(* IEC 61131-3 sources: elnaProjects/ElpcLogic/PomarKc7Changed/build_USO_ecl (part 6) *)

  StrAlg.status :=  SHL(BYTE_TO_DWORD(source_for_Status), 29)
  			OR SHL(BYTE_TO_DWORD(cmd_for_Status), 26)
  			OR SHL(BYTE_TO_DWORD(command_error_for_Status), 23)
  			OR SHL(BOOL_TO_DWORD(StrAlg.OpcCommandsDisabled ), 21)
  			OR SHL(BOOL_TO_DWORD(StrAlg.hasError),4)
  			OR SHL(BOOL_TO_DWORD(StrAlg.CanRun),2)
  			OR SHL(BOOL_TO_DWORD(StrAlg.isEnded),1)
  			OR BOOL_TO_DWORD(StrAlg.isRuning);
END_FUNCTION_BLOCK

FUNCTION_BLOCK fb_AutoTenAlg
  VAR_IN_OUT
    StrAlg : struct_Alg;
    PNS : struct_Switch;
    TEN : struct_Switch;
  END_VAR
  VAR_INPUT
    T_masla : struct_AI;
    Uroven_masla : struct_AI;
    offTemperature : struct_AnalogParametr;
  END_VAR
  VAR
    _sunpackerCommand : fb_sunpackerCommand;
    _statusAi : TYPE_StatusAi;
    _statusDualInput : TYPE_statusDualInput;
    _commandDualInput : TYPE_commandDualInput;
    source : BYTE;
    cmd : BYTE;
    lastCmd : BYTE;
    source_for_Status : BYTE;
    cmd_for_Status : BYTE;
    command_error_for_Status : BYTE;
    resetCmdTimer : TON;
    resetCmdTimerPriznak : BOOL;
    onInit : BOOL;
  END_VAR

  IF NOT onInit THEN
  StrAlg.inCanRun:=TRUE;
  onInit:=TRUE;
  END_IF;

  IF StrAlg.isRuning THEN

  IF ((T_masla.interval >= _statusAi.normal) AND (T_masla.value > offTemperature.Value)) OR
  ((Uroven_masla.interval >= _statusAi.normal) AND (Uroven_masla.value < Uroven_masla.LA)) OR
  (PNS.onStatus=_statusDualInput.STATUS_OFF) THEN

        TEN.inOpcCommandsDisabled:=TRUE;

  	IF TEN.onStatus = _statusDualInput.STATUS_ON THEN
            TEN.inCommand_Alg:=BYTE_TO_WORD(_commandDualInput.CMD_OFF);
  	END_IF;

  ELSIF PNS.onStatus = _statusDualInput.STATUS_ON THEN
        TEN.inOpcCommandsDisabled:=FALSE;
  END_IF;

  END_IF;

  StrAlg.CanRun := StrAlg.inCanRun;
  StrAlg.hasError := TEN.CommandFault OR (T_masla.interval < _statusAi.normal) OR (Uroven_masla.interval < _statusAi.normal);

  StrAlg.OpcCommandsDisabled := StrAlg.inOpcCommandsDisabled;

  (* ---- Если управление с ВУ заблокировано, то  передаем команду из алгоритма ---- *)
  IF StrAlg.inOpcCommandsDisabled THEN
  	StrAlg.inCommand := StrAlg.inCommand_Alg;
  ELSE (* иначе передаем команду с АРМа*)
  	StrAlg.inCommand := StrAlg.inCommand_ARM;
  END_IF;

  _sunpackerCommand(command := StrAlg.inCommand);
  	source := _sunpackerCommand.source;
  	cmd := _sunpackerCommand.cmd;

  IF cmd <> 0 AND lastCmd <> cmd AND (((NOT StrAlg.opcCommandsDisabled) AND source > 0) OR source = 0) then
  	CASE BYTE_TO_INT(cmd) OF
  		(*cmdRun*) 1: 	IF StrAlg.CanRun AND NOT StrAlg.hasError THEN
  					StrAlg.isRuning := TRUE;
  					StrAlg.isEnded := FALSE;
  					(*StrAlg.hasError := FALSE;*)

                                                    (*****************       OnRun       *****************)
                                                    IF StrAlg.inOpcCommandsDisabled THEN
  		                              StrAlg.inOpcCommandsDisabled:=FALSE;
                                                    END_IF;
  					cmd_for_Status := cmd;
  					source_for_Status := source;
  					command_error_for_Status := 0;
  				ELSE
  					StrAlg.isRuning := FALSE;
  					StrAlg.isEnded := FALSE;
  					(*StrAlg.hasError 	:= FALSE;*)

  					cmd_for_Status := 0;
  					source_for_Status := source;
  					command_error_for_Status := cmd;
  				END_IF;
  		(*cmdReset*) 2: 	StrAlg.isRuning := FALSE;
  				StrAlg.isEnded := FALSE;
  				(*StrAlg.hasError 	:= FALSE;*)

                                          (*****************       OnReset       *****************)
                                          TEN.inOpcCommandsDisabled:=TRUE;
                                          TEN.inCommand_Alg:=BYTE_TO_WORD(_commandDualInput.CMD_OFF);

  				cmd_for_Status := cmd;
  				source_for_Status := source;
  				command_error_for_Status := 0;
  	END_CASE;
  	resetCmdTimer(IN := false);
  	resetCmdTimerPriznak := TRUE;
  END_IF;
  lastCmd := cmd;

  resetCmdTimer(IN := resetCmdTimerPriznak, PT := T#5S);
  IF resetCmdTimer.Q THEN
  	resetCmdTimerPriznak := FALSE;
  	source_for_Status := 0;
  	cmd_for_Status := 0;
  	command_error_for_Status := 0;
  END_IF;

  (*TODO: TYPE PROGRAM CODE HERE*)
  StrAlg.status :=  SHL(BYTE_TO_DWORD(source_for_Status), 29)
  			OR SHL(BYTE_TO_DWORD(cmd_for_Status), 26)
  			OR SHL(BYTE_TO_DWORD(command_error_for_Status), 23)
  			OR SHL(BOOL_TO_DWORD(StrAlg.OpcCommandsDisabled ), 21)
  			OR SHL(BOOL_TO_DWORD(StrAlg.hasError),4)
  			OR SHL(BOOL_TO_DWORD(StrAlg.CanRun),2)
  			OR SHL(BOOL_TO_DWORD(StrAlg.isEnded),1)
  			OR BOOL_TO_DWORD(StrAlg.isRuning);
END_FUNCTION_BLOCK

FUNCTION_BLOCK fb_AutoPnsAlg
  VAR_IN_OUT
    StrAlg : struct_Alg;
    Nasos : struct_Switch;
  END_VAR
  VAR_INPUT
    diPlow : struct_singleSignal;
    Poil : struct_AI;
    Ust_Run : struct_AnalogParametr;
    Ust_Stop : struct_AnalogParametr;
  END_VAR
  VAR
    _sunpackerCommand : fb_sunpackerCommand;
    _statusAi : TYPE_StatusAi;
    _statusDualInput : TYPE_statusDualInput;
    _commandDualInput : TYPE_commandDualInput;
    source : BYTE;
    cmd : BYTE;
    lastCmd : BYTE;
    source_for_Status : BYTE;
    cmd_for_Status : BYTE;
    command_error_for_Status : BYTE;
    resetCmdTimer : TON;
    resetCmdTimerPriznak : BOOL;
    onInit : BOOL;
    onTrig : R_TRIG;
    offTrig : R_TRIG;
    waitOn : TON;
    waitOff : TON;
  END_VAR
  VAR_EXTERNAL
    AlgTimers : struct_AlgTimers;
  END_VAR

  IF NOT onInit THEN
  StrAlg.inOpcCommandsDisabled:=TRUE;
  StrAlg.inCanRun:=TRUE;
  onInit:=TRUE;
  END_IF;

  IF StrAlg.isRuning THEN

  StrAlg.hasError := Nasos.CommandFault OR (Poil.interval < _statusAi.normal OR NOT diPlow.reliability);

      IF (Poil.Interval >= _statusAi.normal) THEN
      waitOn(IN:=Poil.Value <= Ust_Run.value OR diPlow.q, PT := T#1S);
      waitOff(IN:= Poil.Value >= Ust_Stop.value, PT := T#300S);

      ELSE
      waitOn(IN:=diPlow.Q, PT := T#1S);
      END_IF;

  onTrig(CLK:=waitOn.Q);
  offTrig(CLK:=waitOff.Q);
      IF (Poil.Value>=Ust_Stop.value) AND Nasos.inopcCommandsDisabled THEN
          Nasos.inopcCommandsDisabled:=FALSE;
      END_IF;

      IF onTrig.Q THEN
      Nasos.inopcCommandsDisabled:=TRUE;
      Nasos.inCommand_Alg:=BYTE_TO_WORD(_commandDualInput.CMD_ON);
      END_IF;

      IF offTrig.Q THEN
          IF NOT (Nasos.onStatus=_statusDualInput.STATUS_OFF) THEN
          Nasos.inopcCommandsDisabled:=TRUE;
          Nasos.inCommand_Alg:=BYTE_TO_WORD(_commandDualInput.CMD_OFF);
          END_IF;
      END_IF;

  AlgTimers.AutoPns_OnTimer:=UDINT_TO_UINT(TIME_TO_UDINT(waitOn.PT - waitOn.ET)/1000);
  AlgTimers.AutoPns_OffTimer:=UDINT_TO_UINT(TIME_TO_UDINT(waitOff.PT -waitOff.ET)/1000);

  END_IF;

  StrAlg.CanRun := StrAlg.inCanRun;

  StrAlg.OpcCommandsDisabled := StrAlg.inOpcCommandsDisabled;

  (* ---- Если управление с ВУ заблокировано, то  передаем команду из алгоритма ---- *)
  IF StrAlg.inOpcCommandsDisabled THEN
  	StrAlg.inCommand := StrAlg.inCommand_Alg;
  ELSE (* иначе передаем команду с АРМа*)
  	StrAlg.inCommand := StrAlg.inCommand_ARM;
  END_IF;

  _sunpackerCommand(command := StrAlg.inCommand);
  	source := _sunpackerCommand.source;
  	cmd := _sunpackerCommand.cmd;

  IF cmd <> 0 AND lastCmd <> cmd AND (((NOT StrAlg.opcCommandsDisabled) AND source > 0) OR source = 0) then
  	CASE BYTE_TO_INT(cmd) OF
  		(*cmdRun*) 1: 	IF (StrAlg.CanRun) THEN
  					StrAlg.isRuning := TRUE;
  					StrAlg.isEnded := FALSE;
  					StrAlg.hasError := FALSE;
  					(*****************       OnRun       *****************)

  					cmd_for_Status := cmd;
  					source_for_Status := source;
  					command_error_for_Status := 0;
  				ELSE
  					StrAlg.isRuning := FALSE;
  					StrAlg.isEnded := FALSE;
  					StrAlg.hasError 	:= FALSE;

  					cmd_for_Status := 0;
  					source_for_Status := source;
  					command_error_for_Status := cmd;
  				END_IF;
  		(*cmdReset*) 2: 	StrAlg.isRuning := FALSE;
  				StrAlg.isEnded := FALSE;
  				StrAlg.hasError 	:= FALSE;

                                           (*****************       OnReset       *****************)
                                          waitOn(in:=FALSE);
                                          waitOff(in:=FALSE);
                                          AlgTimers.AutoPns_OffTimer:=UDINT_TO_UINT(TIME_TO_UDINT(waitOff.pt -waitOff.ET)/1000);

  				cmd_for_Status := cmd;
  				source_for_Status := source;
  				command_error_for_Status := 0;
  	END_CASE;
  	resetCmdTimer(IN := false);
  	resetCmdTimerPriznak := TRUE;
  END_IF;
  lastCmd := cmd;

  resetCmdTimer(IN := resetCmdTimerPriznak, PT := T#5S);
  IF resetCmdTimer.Q THEN
  	resetCmdTimerPriznak := FALSE;
  	source_for_Status := 0;
  	cmd_for_Status := 0;
  	command_error_for_Status := 0;
  END_IF;

  (*TODO: TYPE PROGRAM CODE HERE*)
  StrAlg.status :=  SHL(BYTE_TO_DWORD(source_for_Status), 29)
  			OR SHL(BYTE_TO_DWORD(cmd_for_Status), 26)
  			OR SHL(BYTE_TO_DWORD(command_error_for_Status), 23)
  			OR SHL(BOOL_TO_DWORD(StrAlg.OpcCommandsDisabled ), 21)
  			OR SHL(BOOL_TO_DWORD(StrAlg.hasError),4)
  			OR SHL(BOOL_TO_DWORD(StrAlg.CanRun),2)
  			OR SHL(BOOL_TO_DWORD(StrAlg.isEnded),1)
  			OR BOOL_TO_DWORD(StrAlg.isRuning);
END_FUNCTION_BLOCK

FUNCTION_BLOCK fb_AutoAvomAlg
  VAR_IN_OUT
    StrAlg : struct_Alg;
    im1 : struct_Switch;
    im2 : struct_Switch;
  END_VAR
  VAR_INPUT
    ai : struct_AI;
  END_VAR
  VAR_IN_OUT
    on1Temperature : struct_AnalogParametr;
    on2Temperature : struct_AnalogParametr;
    hystereses : struct_AnalogParametr;
  END_VAR
  VAR
    _sunpackerCommand : fb_sunpackerCommand;
    _statusAi : TYPE_StatusAi;
    _statusDualInput : TYPE_statusDualInput;
    _commandDualInput : TYPE_commandDualInput;
    source : BYTE;
    cmd : BYTE;
    lastCmd : BYTE;
    source_for_Status : BYTE;
    cmd_for_Status : BYTE;
    command_error_for_Status : BYTE;
    resetCmdTimer : TON;
    resetCmdTimerPriznak : BOOL;
    onInit : BOOL;
  END_VAR

  (*
  IF NOT onInit THEN
  StrAlg.inCanRun:=TRUE;
  onInit:=TRUE;
  END_IF;
  *)

  IF StrAlg.isRuning THEN

  StrAlg.hasError := im1.CommandFault OR im2.CommandFault OR (ai.interval<_statusAi.normal);

      IF (ai.interval>=_statusAi.normal) THEN

            IF (ai.value>= on1Temperature.Value) THEN
                IF im1.onStatus <> _statusDualInput.STATUS_ON THEN
  	       im1.inCommand_Alg:=BYTE_TO_WORD(_commandDualInput.CMD_ON); (*cmd_on*)
                END_IF;
            END_IF;

            IF  ai.value < (on1Temperature.Value - hystereses.Value) THEN
                IF im1.onStatus <> _statusDualInput.STATUS_OFF THEN
  	       im1.inCommand_Alg:=BYTE_TO_WORD(_commandDualInput.CMD_OFF);
                END_IF;
            END_IF;

             IF (ai.value>= on2Temperature.Value) THEN
                IF im2.onStatus <> _statusDualInput.STATUS_ON THEN
  	       im2.inCommand_Alg:=BYTE_TO_WORD(_commandDualInput.CMD_ON); (*cmd_on*)
                END_IF;
            END_IF;

            IF  ai.value < (on2Temperature.Value - hystereses.Value) THEN
                IF im2.onStatus <> _statusDualInput.STATUS_OFF THEN
  	       im2.inCommand_Alg:=BYTE_TO_WORD(_commandDualInput.CMD_OFF);
                END_IF;
            END_IF;
       END_IF;

  END_IF;

  StrAlg.CanRun := StrAlg.inCanRun;

  StrAlg.OpcCommandsDisabled := StrAlg.inOpcCommandsDisabled;

  (* ---- Если управление с ВУ заблокировано, то  передаем команду из алгоритма ---- *)
  IF StrAlg.inOpcCommandsDisabled THEN
  	StrAlg.inCommand := StrAlg.inCommand_Alg;
  ELSE (* иначе передаем команду с АРМа*)
  	StrAlg.inCommand := StrAlg.inCommand_ARM;
  END_IF;

  _sunpackerCommand(command := StrAlg.inCommand);
  	source := _sunpackerCommand.source;
  	cmd := _sunpackerCommand.cmd;

  IF cmd <> 0 AND lastCmd <> cmd AND (((NOT StrAlg.opcCommandsDisabled) AND source > 0) OR source = 0) then
  	CASE BYTE_TO_INT(cmd) OF
  		(*cmdRun*) 1: 	IF (StrAlg.CanRun) THEN
  					StrAlg.isRuning := TRUE;
  					StrAlg.isEnded := FALSE;
  					StrAlg.hasError := FALSE;
                                                    StrAlg.inOpcCommandsDisabled:=FALSE;
  					im1.inOpcCommandsDisabled:=TRUE;
                                                    im2.inOpcCommandsDisabled:=TRUE;
  					cmd_for_Status := cmd;
  					source_for_Status := source;
  					command_error_for_Status := 0;
  				ELSE
  					StrAlg.isRuning := FALSE;
  					StrAlg.isEnded := FALSE;
  					StrAlg.hasError 	:= FALSE;

  					cmd_for_Status := 0;
  					source_for_Status := source;
  					command_error_for_Status := cmd;
  				END_IF;
  		(*cmdReset*) 2: 	StrAlg.isRuning := FALSE;
  				StrAlg.isEnded := FALSE;
  				StrAlg.hasError 	:= FALSE;
                                          StrAlg.inOpcCommandsDisabled:=FALSE;
                                          im1.inOpcCommandsDisabled:=FALSE;
                                          im2.inOpcCommandsDisabled:=FALSE;
                                          im1.inCommand_Alg:=0;
                                          im2.inCommand_Alg:=0;
  				cmd_for_Status := cmd;
  				source_for_Status := source;
  				command_error_for_Status := 0;
  	END_CASE;
  	resetCmdTimer(IN := false);
  	resetCmdTimerPriznak := TRUE;
  END_IF;
  lastCmd := cmd;

  resetCmdTimer(IN := resetCmdTimerPriznak, PT := T#5S);
  IF resetCmdTimer.Q THEN
  	resetCmdTimerPriznak := FALSE;
  	source_for_Status := 0;
  	cmd_for_Status := 0;
  	command_error_for_Status := 0;
  END_IF;

  (*TODO: TYPE PROGRAM CODE HERE*)
  StrAlg.status :=  SHL(BYTE_TO_DWORD(source_for_Status), 29)
  			OR SHL(BYTE_TO_DWORD(cmd_for_Status), 26)
  			OR SHL(BYTE_TO_DWORD(command_error_for_Status), 23)
  			OR SHL(BOOL_TO_DWORD(StrAlg.OpcCommandsDisabled ), 21)
  			OR SHL(BOOL_TO_DWORD(StrAlg.hasError),4)
  			OR SHL(BOOL_TO_DWORD(StrAlg.CanRun),2)
  			OR SHL(BOOL_TO_DWORD(StrAlg.isEnded),1)
  			OR BOOL_TO_DWORD(StrAlg.isRuning);
END_FUNCTION_BLOCK

FUNCTION_BLOCK fb_vibegPNSAlg
  VAR_IN_OUT
    StrAlg : struct_Alg;
  END_VAR
  VAR
    autoPnsOff : struct_PhaseAlgoritm;
    waitVibeg : struct_PhaseAlgoritm;
    pnsOff : struct_PhaseAlgoritm;
    vibegEnd : struct_PhaseAlgoritm;
  END_VAR
  VAR_IN_OUT
    algContinue : struct_Question;
  END_VAR
  VAR
    fb_autoPnsOff : fb_ph_algoritm;
    fb_waitVibeg : fb_ph_Timer;
    fb_algContinue : fb_Question;
    fb_pnsOff : fb_ph_Switch;
    fb_vibegEnd : fb_ph_CustomPhase;
    _sunpackerCommand : fb_sunpackerCommand;
    _statusAi : TYPE_StatusAi;
    _Answers : TYPE_Answers;
    _statusDualInput : TYPE_statusDualInput;
    _DualStateImAction : TYPE_DualStateImAction;
    _PhaseAlgoritmAction : TYPE_PhaseAlgoritmAction;
    source : BYTE;
    cmd : BYTE;
    lastCmd : BYTE;
    source_for_Status : BYTE;
    cmd_for_Status : BYTE;
    command_error_for_Status : BYTE;
    resetCmdTimer : TON;
    resetCmdTimerPriznak : BOOL;
    onInit : BOOL;
    waitReset : TON;
  END_VAR
  VAR_EXTERNAL
    IM : ImConfig;
    algoritms : AlgoritmsConfig;
    ai : AiConfig;
    protections : ProtectionsConfig;
    AlgTimers : struct_AlgTimers;
  END_VAR

  IF NOT onInit THEN
   fb_autoPnsOff(phaseNumber:=0, act:=_reset, waitCompletion:=FALSE);
    fb_waitVibeg(phaseNumber:=1, delay:=T#300S);
       algContinue.AnswerVariants:=_Answers.ANS_YES;
       fb_pnsOff(phaseNumber:=2, act:=_off);
     fb_vibegEnd(phaseNumber:=14);
  onInit:=TRUE;
  END_IF;

   fb_autoPnsOff(StrPh:=autoPnsOff, alg:=algoritms.autoPns);
    fb_waitVibeg(StrPh:=waitVibeg, timer:=AlgTimers.vibegPNS_Timer);
  fb_algContinue(StrQ:=algContinue);
       fb_pnsOff(StrPh:=pnsOff, Im:=IM.pns);
     fb_vibegEnd(StrPh:=vibegEnd);

  IF StrAlg.isRuning THEN

  StrAlg.hasError := autoPnsOff.error OR pnsOff.error;

      IF IM.pns.onStatus = _statusDualInput.STATUS_ON AND NOT vibegEnd.top THEN

  	runPhase(vibegEnd);
            runPhase(waitVibeg);
            askQuestion(algContinue);

      END_IF;

      IF waitVibeg.top OR (algContinue.answer = _Answers.ANS_YES) THEN
  	vibegEnd.top:=TRUE;
  	resetPhase(waitVibeg);
            resetQuestion(algContinue);

            resetAiProtection(protections.Os_sdvig_nagnetatelja_minus);
            (*resetDiProtection(protections.Vibro_skorost_OP_shesterni_RED_T6);*)

  	(*IM.SingleSignals.P_oil_low.Disabled_Sig:=TRUE;*)
  	ai.Pmasla_posle_GNS.Disabled_LA:=TRUE;
            ai.Pmasla_posle_GNS.Disabled_LW:=TRUE;
            ai.Pmasla_posle_NU.Disabled_LW:=TRUE;
  	runPhase(pnsOff);
      END_IF;

      StrAlg.isEnded:=pnsOff.top;

  END_IF;

  StrAlg.CanRun := StrAlg.inCanRun;
  StrAlg.OpcCommandsDisabled := StrAlg.inOpcCommandsDisabled;

  (* ---- Если управление с ВУ заблокировано, то  передаем команду из алгоритма ---- *)
  IF StrAlg.inOpcCommandsDisabled THEN
  	StrAlg.inCommand := StrAlg.inCommand_Alg;
  ELSE (* иначе передаем команду с АРМа*)
  	StrAlg.inCommand := StrAlg.inCommand_ARM;
  END_IF;

  _sunpackerCommand(command := StrAlg.inCommand);
  	source := _sunpackerCommand.source;
  	cmd := _sunpackerCommand.cmd;

  IF cmd <> 0 AND lastCmd <> cmd AND (((NOT StrAlg.opcCommandsDisabled) AND source > 0) OR source = 0) then
  	CASE BYTE_TO_INT(cmd) OF
  		(*cmdRun*) 1: 	IF (StrAlg.CanRun) THEN
  					StrAlg.isRuning := TRUE;
  					StrAlg.isEnded := FALSE;
  					StrAlg.hasError := FALSE;
  					(*****************       OnRun       *****************)
                                                    runPhase(autoPnsOff);

  					cmd_for_Status := cmd;
  					source_for_Status := source;
  					command_error_for_Status := 0;
  				ELSE
  					StrAlg.isRuning := FALSE;
  					StrAlg.isEnded := FALSE;
  					StrAlg.hasError 	:= FALSE;

  					cmd_for_Status := 0;
  					source_for_Status := source;
  					command_error_for_Status := cmd;
  				END_IF;
  		(*cmdReset*) 2: 	StrAlg.isRuning := FALSE;
  				StrAlg.isEnded := FALSE;
  				StrAlg.hasError 	:= FALSE;

                                           (*****************       OnReset       *****************)
                                         waitReset(IN:=FALSE);
                                         resetPhase(autoPnsOff);
                                         resetPhase(waitVibeg);
                                         resetPhase(vibegEnd);
                                         resetPhase(pnsOff);
                                         resetQuestion(algContinue);

  				cmd_for_Status := cmd;
  				source_for_Status := source;
  				command_error_for_Status := 0;
  	END_CASE;
  	resetCmdTimer(IN := false);
  	resetCmdTimerPriznak := TRUE;
  END_IF;
  lastCmd := cmd;

  resetCmdTimer(IN := resetCmdTimerPriznak, PT := T#5S);
  IF resetCmdTimer.Q THEN
  	resetCmdTimerPriznak := FALSE;
  	source_for_Status := 0;
  	cmd_for_Status := 0;
  	command_error_for_Status := 0;
  END_IF;

  StrAlg.Start:= autoPnsOff.startStatus
              OR waitVibeg.startStatus
              OR pnsOff.startStatus
              OR vibegEnd.startStatus;

  StrAlg.Error:= autoPnsOff.errorStatus
              OR waitVibeg.errorStatus
              OR pnsOff.errorStatus
              OR vibegEnd.errorStatus;

  StrAlg.Top:=   autoPnsOff.topStatus
              OR waitVibeg.topStatus
              OR pnsOff.topStatus
              OR vibegEnd.topStatus;

  (*TODO: TYPE PROGRAM CODE HERE*)
  StrAlg.status :=  SHL(BYTE_TO_DWORD(source_for_Status), 29)
  			OR SHL(BYTE_TO_DWORD(cmd_for_Status), 26)
  			OR SHL(BYTE_TO_DWORD(command_error_for_Status), 23)
  			OR SHL(BOOL_TO_DWORD(StrAlg.OpcCommandsDisabled ), 21)
  			OR SHL(BOOL_TO_DWORD(StrAlg.hasError),4)
  			OR SHL(BOOL_TO_DWORD(StrAlg.CanRun),2)
  			OR SHL(BOOL_TO_DWORD(StrAlg.isEnded),1)
  			OR BOOL_TO_DWORD(StrAlg.isRuning);
END_FUNCTION_BLOCK

FUNCTION_BLOCK fb_AutoNUAlg
  VAR_IN_OUT
    StrAlg : struct_Alg;
    nu1 : struct_OilPump;
    nu2 : struct_OilPump;
  END_VAR
  VAR_INPUT
    dPoil : struct_AI;
  END_VAR
  VAR_IN_OUT
    mainNU : struct_DiscretParametr;
    Lowdp_di : struct_singleSignal;
    Ust_Swap : struct_AnalogParametr;
  END_VAR
  VAR
    _prevMainNU : UINT;
    _sunpackerCommand : fb_sunpackerCommand;
    _statusAi : TYPE_StatusAi;
    _statusDualInput : TYPE_statusDualInput;
    _commandDualInput : TYPE_commandDualInput;
    source : BYTE;
    cmd : BYTE;
    lastCmd : BYTE;
    source_for_Status : BYTE;
    cmd_for_Status : BYTE;
    command_error_for_Status : BYTE;
    resetCmdTimer : TON;
    waitPressure : TON;
    waitPressureTrig : R_TRIG;
    resetCmdTimerPriznak : BOOL;
    onInit : BOOL;
    onStart : BOOL;
  END_VAR
  VAR_EXTERNAL
    NotHasRezervNU : BOOL;
    Reset_HasNU : BOOL;
  END_VAR

  IF NOT onInit THEN
  StrAlg.inCanRun:=TRUE;
  StrAlg.inOpcCommandsDisabled:=TRUE;
  (*nu1.Osnovnoy:=TRUE; nu2.Osnovnoy:=FALSE;*)
  onInit:=TRUE;
  END_IF;

  IF Reset_HasNU THEN
  nu1.inBlocked:=FALSE;
  nu2.inBlocked:=FALSE;
  END_IF;

  NotHasRezervNU:=(nu1.Blocked OR nu2.Blocked);

  IF StrAlg.isRuning THEN

  StrAlg.hasError := nu1.CommandFault OR nu2.CommandFault OR (dPoil.interval<_statusAi.normal);

   IF mainNU.value<>_prevMainNU OR NOT onStart THEN

          CASE mainNU.value OF
  	0: nu1.Osnovnoy:=TRUE; nu2.Osnovnoy:=FALSE;
  	1: nu1.Osnovnoy:=FALSE; nu2.Osnovnoy:=TRUE;

          END_CASE;

      IF  nu1.Osnovnoy AND NOT nu1.Blocked THEN
          nu1.inCommand_Alg:=BYTE_TO_WORD(_commandDualInput.CMD_ON);
      ELSIF NOT NotHasRezervNU THEN
          nu1.inCommand_Alg:=BYTE_TO_WORD(_commandDualInput.CMD_OFF);
      END_IF;

      IF  nu2.Osnovnoy AND NOT nu2.Blocked THEN
          nu2.inCommand_Alg:=BYTE_TO_WORD(_commandDualInput.CMD_ON);
       ELSIF NOT NotHasRezervNU THEN
          nu2.inCommand_Alg:=BYTE_TO_WORD(_commandDualInput.CMD_OFF);
      END_IF;
        onStart:=TRUE;
       _prevMainNU:=mainNU.value;
   END_IF;

    (*IF (nu1.onStatus = _statusDualInput.STATUS_On) OR (nu2.onStatus = _statusDualInput.STATUS_On) THEN*)
      (*Если через 5С насос не нагнал 100кПа масла - он сломался и надо переключить насос*)
      IF dPoil.interval>= _statusAi.NORMAL THEN
            waitPressure(IN:=(dPoil.value<Ust_Swap.Value OR LowdP_DI.q) AND NOT NotHasRezervNU, PT:= T#5S);
      ELSE
  	waitPressure(IN:=(FALSE));
      END_IF;

      waitPressureTrig(CLK:=waitPressure.Q);
      IF waitPressureTrig.Q THEN
  	(*IF nu1.onStatus = _statusDualInput.STATUS_ON THEN*)
             IF mainNU.value = 0 THEN
  		nu1.inBlocked:=TRUE;
                      nu1.inCommand_Alg:=BYTE_TO_WORD(_commandDualInput.CMD_OFF);
  			(*IF 	mainNU.value = 0 THEN*)
                                          setValue(mainNU, 1);
  			(*END_IF;*)
  	END_IF;

  	(*IF nu2.onStatus = _statusDualInput.STATUS_ON THEN*)
            IF mainNU.value = 1 THEN
  		nu2.inBlocked:=TRUE;
                      nu2.inCommand_Alg:=BYTE_TO_WORD(_commandDualInput.CMD_OFF);
  			(*IF 	mainNU.value = 1 THEN*)
  				setValue(mainNU, 0);
  			(*END_IF;*)
  	END_IF;
      END_IF;
   (* END_IF;*)

  END_IF;

  StrAlg.CanRun := StrAlg.inCanRun;

  StrAlg.OpcCommandsDisabled := StrAlg.inOpcCommandsDisabled;

  (* ---- Если управление с ВУ заблокировано, то  передаем команду из алгоритма ---- *)
  IF StrAlg.inOpcCommandsDisabled THEN
  	StrAlg.inCommand := StrAlg.inCommand_Alg;
  ELSE (* иначе передаем команду с АРМа*)
  	StrAlg.inCommand := StrAlg.inCommand_ARM;
  END_IF;

  _sunpackerCommand(command := StrAlg.inCommand);
  	source := _sunpackerCommand.source;
  	cmd := _sunpackerCommand.cmd;

  IF cmd <> 0 AND lastCmd <> cmd AND (((NOT StrAlg.opcCommandsDisabled) AND source > 0) OR source = 0) then
  	CASE BYTE_TO_INT(cmd) OF
  		(*cmdRun*) 1: 	IF (StrAlg.CanRun) THEN
  					StrAlg.isRuning := TRUE;
  					StrAlg.isEnded := FALSE;
  					StrAlg.hasError := FALSE;

                                                    (*****************       OnRun       *****************)
  					nu1.inOpcCommandsDisabled:=TRUE;
                                                    nu2.inOpcCommandsDisabled:=TRUE;

  					cmd_for_Status := cmd;
  					source_for_Status := source;
  					command_error_for_Status := 0;
  				ELSE
  					StrAlg.isRuning := FALSE;
  					StrAlg.isEnded := FALSE;
  					StrAlg.hasError 	:= FALSE;

  					cmd_for_Status := 0;
  					source_for_Status := source;
  					command_error_for_Status := cmd;
  				END_IF;
  		(*cmdReset*) 2: 	StrAlg.isRuning := FALSE;
  				StrAlg.isEnded := FALSE;
  				StrAlg.hasError 	:= FALSE;

                                          (*****************       OnReset       *****************)
                                          waitPressure(IN:=(FALSE));
                                          onStart:=FALSE;

  				cmd_for_Status := cmd;
  				source_for_Status := source;
  				command_error_for_Status := 0;
  	END_CASE;
  	resetCmdTimer(IN := false);
  	resetCmdTimerPriznak := TRUE;
  END_IF;
  lastCmd := cmd;

  resetCmdTimer(IN := resetCmdTimerPriznak, PT := T#5S);
  IF resetCmdTimer.Q THEN
  	resetCmdTimerPriznak := FALSE;
  	source_for_Status := 0;
  	cmd_for_Status := 0;
  	command_error_for_Status := 0;
  END_IF;

  (*TODO: TYPE PROGRAM CODE HERE*)
  StrAlg.status :=  SHL(BYTE_TO_DWORD(source_for_Status), 29)
  			OR SHL(BYTE_TO_DWORD(cmd_for_Status), 26)
  			OR SHL(BYTE_TO_DWORD(command_error_for_Status), 23)
  			OR SHL(BOOL_TO_DWORD(StrAlg.OpcCommandsDisabled ), 21)
                                OR SHL(BOOL_TO_DWORD(NotHasRezervNU), 15)
  			OR SHL(BOOL_TO_DWORD(StrAlg.hasError),4)
  			OR SHL(BOOL_TO_DWORD(StrAlg.CanRun),2)
  			OR SHL(BOOL_TO_DWORD(StrAlg.isEnded),1)
  			OR BOOL_TO_DWORD(StrAlg.isRuning);
END_FUNCTION_BLOCK

FUNCTION_BLOCK AOAlg
  VAR_IN_OUT
    StrAlg : struct_Alg;
  END_VAR
  VAR
    kran6Open : struct_PhaseAlgoritm;
    kran4Close : struct_PhaseAlgoritm;
    kran3bOpen : struct_PhaseAlgoritm;
    mvOff : struct_PhaseAlgoritm;
    kran1Close : struct_PhaseAlgoritm;
    kran2Close : struct_PhaseAlgoritm;
    kran3Close : struct_PhaseAlgoritm;
    kran5Open : struct_PhaseAlgoritm;
    autoPnsOff : struct_PhaseAlgoritm;
    pnsOn : struct_PhaseAlgoritm;
    Pg_VhodLessThen300 : struct_PhaseAlgoritm;
    Pg_VyhodLessThen300 : struct_PhaseAlgoritm;
    nu1off : struct_PhaseAlgoritm;
    nu2off : struct_PhaseAlgoritm;
    AutoNU_Off : struct_PhaseAlgoritm;
    timer600 : struct_PhaseAlgoritm;
    pnsOff : struct_PhaseAlgoritm;
    Avom1Off : struct_PhaseAlgoritm;
    Avom2Off : struct_PhaseAlgoritm;
    Avom3Off : struct_PhaseAlgoritm;
    Avom4Off : struct_PhaseAlgoritm;
    autoAVOMOff : struct_PhaseAlgoritm;
    timer5 : struct_PhaseAlgoritm;
    klapan1 : struct_PhaseAlgoritm;
    klapan2 : struct_PhaseAlgoritm;
    nu_On : struct_PhaseAlgoritm;
    Start_AO_From : struct_PhaseAlgoritm;
    fb_kran6Open : fb_ph_Kran;
    fb_pnsOn : fb_ph_Switch;
    fb_kran4Close : fb_ph_Kran;
    fb_kran3bOpen : fb_ph_Kran;
    fb_mvOff : fb_ph_SectionSwitch;
    fb_kran1Close : fb_ph_Kran;
    fb_kran2Close : fb_ph_Kran;
    fb_kran3Close : fb_ph_Kran;
    fb_kran5Open : fb_ph_Kran;
    fb_autoPnsOff : fb_ph_algoritm;
    fb_Pg_VhodLessThen300 : fb_ph_CustomPhase;
    fb_Pg_VyhodLessThen300 : fb_ph_CustomPhase;
    fb_nu1Off : fb_ph_OilPump;
    fb_nu2Off : fb_ph_OilPump;
    fb_autoNuOff : fb_ph_algoritm;
    fb_timer600 : fb_ph_Timer;
    fb_pnsOff : fb_ph_Switch;
    fb_Avom1Off : fb_ph_Switch;
    fb_Avom2Off : fb_ph_Switch;
    fb_Avom3Off : fb_ph_Switch;
    fb_Avom4Off : fb_ph_Switch;
    fb_autoAVOMOff : fb_ph_algoritm;
    fb_timer5 : fb_ph_Timer;
    fb_klapan1 : fb_ph_CustomPhase;
    fb_klapan2 : fb_ph_CustomPhase;
    fb_nu_On : fb_ph_CustomPhase;
    fb_Start_AO_From : fb_ph_CustomPhase;
    _sunpackerCommand : fb_sunpackerCommand;
    _statusAi : TYPE_StatusAi;
    _Answers : TYPE_Answers;
    _statusDualInput : TYPE_statusDualInput;
    _commandDualInput : TYPE_commandDualInput;
    _DualStateImAction : TYPE_DualStateImAction;
    _PhaseAlgoritmAction : TYPE_PhaseAlgoritmAction;
    source : BYTE;
    cmd : BYTE;
    lastCmd : BYTE;
    source_for_Status : BYTE;
    cmd_for_Status : BYTE;
    command_error_for_Status : BYTE;
    resetCmdTimer : TON;
    resetCmdTimerPriznak : BOOL;
    onInit : BOOL;
    waitReset : TON;
  END_VAR
  VAR_EXTERNAL
    IM : ImConfig;
    algoritms : AlgoritmsConfig;
    ai : AiConfig;
    protections : ProtectionsConfig;
    ModeGpa : TYPE_ModeGpa;
    algManager : struct_AlgoritmsManager;
    AlgTimers : struct_AlgTimers;
  END_VAR
  VAR CONSTANT
    Ust_Pgaza : LREAL          := 0.3;
  END_VAR

  IF NOT onInit THEN
      fb_kran6Open(phaseNumber:=1, act:=_on);
      fb_kran4Close(phaseNumber:=2, act:=_off);
      fb_kran3bOpen(phaseNumber:=3, act:=_off);
      fb_mvOff(phaseNumber:=4, act:=_off);
      fb_kran1Close(phaseNumber:=5, act:=_off);
      fb_kran2Close(phaseNumber:=6, act:=_off);
      fb_kran3Close(phaseNumber:=7, act:=_off);
      fb_kran5Open(phaseNumber:=8, act:=_on);
      fb_autoPnsOff(phaseNumber:=9, act:=_reset, waitCompletion:=FALSE);
      fb_pnsOn(phaseNumber:=10, act:=_on);
      fb_Pg_VhodLessThen300(phaseNumber:=11);
      fb_Pg_VyhodLessThen300(phaseNumber:=12);
      fb_nu1Off(phaseNumber:=13, act:=_off);
      fb_nu2Off(phaseNumber:=14, act:=_off);
      fb_autoNuOff(phaseNumber:=15, act:=_reset, waitCompletion:=FALSE);
      fb_timer600(phaseNumber:=16, delay:=T#600S);
      fb_pnsOff(phaseNumber:=17, act:=_off);
      fb_Avom1Off(phaseNumber:=18, act:=_off);
      fb_Avom2Off(phaseNumber:=19, act:=_off);
      fb_Avom3Off(phaseNumber:=20, act:=_off);
      fb_Avom4Off(phaseNumber:=21, act:=_off);
      fb_autoAVOMOff(phaseNumber:=22, act:=_reset, waitCompletion:=FALSE);
      fb_timer5(phaseNumber:=23, delay:=T#5S);
      fb_klapan1(phaseNumber:=24);
      fb_klapan2(phaseNumber:=25);
      fb_nu_On(phaseNumber:=26);
      fb_Start_AO_From(phaseNumber:=27);
  onInit:=TRUE;
  END_IF;

  fb_kran6Open(StrPh:=kran6Open, Im:=Im.kran6);
  fb_pnsOn(StrPh:=pnsOn, Im:=Im.pns);
  fb_kran4Close(StrPh:=kran4Close, Im:=Im.kran4);
  fb_kran3bOpen(StrPh:=kran3bOpen, Im:=Im.kran3b);
  fb_mvOff(StrPh:=mvOff, Im:=Im.mv);
  fb_kran1Close(StrPh:=kran1Close, Im:=Im.kran1);
  fb_kran2Close(StrPh:=kran2Close, Im:=Im.Kran2);
  fb_kran3Close(StrPh:=kran3Close, Im:=Im.Kran3);
  fb_kran5Open(StrPh:=kran5Open, Im:=Im.Kran5);
  fb_autoPnsOff(StrPh:=autoPnsOff, alg:=algoritms.autoPns);
  fb_Pg_VhodLessThen300(StrPh:=Pg_VhodLessThen300);
  fb_Pg_VyhodLessThen300(StrPh:=Pg_VyhodLessThen300);
  fb_nu1Off(StrPh:=nu1off, Im:=Im.nu1);
  fb_nu2Off(StrPh:=nu2off, Im:=Im.nu2);
  fb_autoNuOff(StrPh:=AutoNU_Off, alg:=algoritms.autoNu);
  fb_timer600(StrPh:=timer600, timer:=AlgTimers.No_wait600);
  fb_pnsOff(StrPh:=pnsOff, Im:=Im.pns);
  fb_Avom1Off(StrPh:=Avom1Off, Im:=Im.v1_Avom);
  fb_Avom2Off(StrPh:=Avom2Off, Im:=Im.v2_Avom);
  fb_Avom3Off(StrPh:=Avom3Off, Im:=Im.v3_Avom);
  fb_Avom4Off(StrPh:=Avom4Off, Im:=Im.v4_Avom);
  fb_autoAVOMOff(StrPh:=autoAVOMOff, alg:=algoritms.AutoAvom);
  fb_timer5(StrPh:=timer5, timer:=AlgTimers.No_wait5);
  fb_klapan1(StrPh:=klapan1);
  fb_klapan2(StrPh:=klapan2);
  fb_nu_On(StrPh:=nu_On);
  fb_Start_AO_From(StrPh:=Start_AO_From);

  StrAlg.CanRun := StrAlg.inCanRun;
  StrAlg.OpcCommandsDisabled := StrAlg.inOpcCommandsDisabled;

  IF StrAlg.isRuning THEN

      IF	(*algoritms.F3.Smazka_1_2 OR*) IM.kran1.onStatus = _statusDualInput.STATUS_ON OR IM.kran1.onStatus = _statusDualInput.STATUS_TRANSITIONAL
  	    OR IM.kran2.onStatus = _statusDualInput.STATUS_ON OR IM.kran2.onStatus = _statusDualInput.STATUS_TRANSITIONAL  THEN
  	    IF (*(algoritms.F3.Smazka_1_2 OR*) IM.kran1.onStatus = _statusDualInput.STATUS_ON OR IM.kran1.onStatus = _statusDualInput.STATUS_TRANSITIONAL AND NOT klapan1.start AND NOT kran1Close.top THEN
  		    runPhase(klapan1);
  	    END_IF;
  	    IF (*algoritms.F3.Smazka_1_2 OR*) IM.kran2.onStatus = _statusDualInput.STATUS_ON OR IM.kran2.onStatus = _statusDualInput.STATUS_TRANSITIONAL AND NOT klapan2.start AND NOT kran2Close.top THEN
  		    runPhase(klapan2);
      	END_IF;
  	(*algoritms.F3.Smazka_1_2:=FALSE; у меня нет такой штуки*)
      END_IF;

     (* IF NOT kran6Open.start THEN
  	    ystavki.Block_kr6_alg.setValue (1);
  	    IF IM.kran6._cmdreset.IN = FALSE THEN
  		    ystavki.Block_kr6_alg.setValue (0); такой штуки тоже нет
  		        runPhase(kran6Open);
  	    END_IF;
      END_IF;*)

      (*IF NOT kran4Close.start THEN
  	    ystavki.Block_kr4_alg.setValue (1);
  	    IF IM.kran4._cmdreset.IN = FALSE THEN
  		    ystavki.Block_kr4_alg.setValue (0);
  		    kran4Close.run();
  	    END_IF;
      END_IF;*)

      (*IF NOT kran3bOpen.start THEN
  	    ystavki.Block_kr3b_alg.setValue (1);
  	    IF IM.kran3b._cmdreset.IN = FALSE THEN
  		    ystavki.Block_kr3b_alg.setValue (0);
  		    runPhase(kran3bOpen);
  	    END_IF;
      END_IF;*)

      resetDiProtection(protections.mvOff);
      resetDiProtection(protections.Off_avar_vikluchatel);
      resetDiProtection(protections.Reg_vozb_off);
      resetDiProtection(protections.Kran1_sdvig);
      resetDiProtection(protections.Kran2_sdvig);
      runPhase(mvOff);

      (*IF NOT kran1Close.start THEN
  	ystavki.Block_kr1_alg.setValue (1);*)
  	    (*IF IM.kran1._cmdreset.IN = FALSE THEN
  		    ystavki.Block_kr1_alg.setValue (0);
  		    runPhase(kran1Close);
  	    END_IF;
      END_IF;*)

      (*IF NOT kran2Close.start THEN
  	    ystavki.Block_kr2_alg.setValue (1);
  	    IF IM.kran2._cmdreset.IN = FALSE THEN
  		    ystavki.Block_kr2_alg.setValue (0);
  		    runPhase(kran2Close);
  	    END_IF;
      END_IF;*)

      (*IF NOT kran3Close.start THEN
  	    ystavki.Block_kr3_alg.setValue (1);
  	    IF	IM.kran3._cmdreset.IN = FALSE THEN
  		    ystavki.Block_kr3_alg.setValue (0);
  		    runPhase(kran3Close);
  	    END_IF;
      END_IF;*)

      (*IF kran6Open.top THEN
  	    algoritms.S_Vibr.CanRun:=FALSE;
  	    algoritms.S_Vibr.reset ();
      END_IF;*)

      IF klapan1.start AND kran1Close.top THEN
  	    (*IM.Kr1_Smazka.impulse();*)
  	    klapan1.top:=TRUE;
      END_IF;
      IF	klapan2.start AND kran2Close.top THEN
  	    (*zIM.Kr2_Smazka.impulse();*)
  	    klapan2.top:=TRUE;
      END_IF;

      (*IF 	kran1Close.top AND kran2Close.top AND kran3Close.top AND kran4Close.top AND NOT kran5Open.top THEN
  	    IF	NOT	kran5Open.start THEN
              ystavki.Block_kr5_alg.setValue (1);
  		    IF	IM.kran5._cmdreset.IN = FALSE THEN
  			    ystavki.Block_kr5_alg.setValue (0);
  			    runPhase(kran5Open);
  		    END_IF;
  	    END_IF;

  	    resetAiProtection(protections.Pgaza_na_vyhode_nagnetatelia);
      END_IF; *)

      IF mvOff.top (*AND NOT flag1*) THEN
  	    (*algoritms.AutoPNS_Start.canrun :=FALSE;
  	    algoritms.AutoPNS_Start.reset ();*)
  	    algoritms.autoPns.canrun :=FALSE;
  	    runPhase(autoPnsOff);
  	    runPhase(pnsOn);
  	    runPhase(nu_On);
  	    (*vkluchit nasosi*)
  	    algoritms.autoNu.canrun:=FALSE;
  	    (*algoritms.autoNu_2.reset ();
  	    algoritms.autoNu_1.canrun:=TRUE;
  	    algoritms.autoNu_1.run ();
  	    flag1:=TRUE;*)
      END_IF;

      IF	IM.nu1.onStatus =_statusDualInput.STATUS_ON OR IM.nu2.onStatus =_statusDualInput.STATUS_ON AND nu_On.start AND NOT nu_On.top THEN
  	    nu_On.top:=TRUE;
      END_IF;

      IF kran5Open.top THEN
  	    runPhase(Pg_VhodLessThen300);
  	    runPhase(Pg_VyhodLessThen300);
  	END_IF;

      IF Pg_VhodLessThen300.start AND NOT Pg_VhodLessThen300.top THEN
  	    IF ai.Pgaza_na_vhode_nagnetatelia.interval >= _statusAi.NORMAL AND ai.Pgaza_na_vhode_nagnetatelia.value < 0.3 THEN
  		    Pg_VhodLessThen300.top:=TRUE;
  	    END_IF;
      END_IF;

      IF Pg_VyhodLessThen300.start AND NOT Pg_VyhodLessThen300.top THEN
  	    IF ai.Pgaza_na_vyhode_nagnetatelia.interval>=_statusAi.NORMAL AND ai.Pgaza_na_vyhode_nagnetatelia.value < 0.3 THEN
  		    Pg_VyhodLessThen300.top:=TRUE;
  	    END_IF;
      END_IF;

      IF Pg_VhodLessThen300.top AND Pg_VyhodLessThen300.top AND pnsOn.top AND nu_On.top AND mvOff.top THEN
  	    runPhase(nu1Off);
      	    resetAiProtection(protections.dPmaslo_gaz);
  	    resetDiProtection(protections.dPmaslo_gaz_less100);
  	    runAiProtection(protections.Pgaza_na_vhode_nagnetatelia_GPA_STOP);
  	    runAiProtection(protections.Pgaza_na_vyhode_nagnetatelia_GPA_STOP);
  	    AutoNU_Off.top:=TRUE;
      	(*algoritms.autoNu_1.CanRun:=FALSE;
  	    algoritms.autoNu_1.reset ();*)
      END_IF;

      (*IF nuOff.top THEN
  	    IF NOT algmanager.reg_V AND NOT pnsoff.start THEN
  		    runPhase(timer600);
  	    END_IF;
  	    IF	NOT pnsoff.start THEN
  		    sbrosVibeg.ask();
  	    END_IF;
      END_IF;*)

      IF timer600.top (*OR sbrosVibeg.answer=Answers.ANS_YES*)  THEN
  	    runPhase(pnsOff);
  	    resetAiProtection(protections.Pmaslo_sm_nizkoe);
  	    resetAiProtection(protections.Pmaslo_sm_vysokoe);
  	    (*resetPhase(sbrosVibeg);*)
  	    resetPhase(timer600);
  	    (*algoritms.F2_Ch.autoAVOM_canrun_flag:=FALSE;
  	    algoritms.F2_R.autoAVOM_canrun_flag:=FALSE;*)
      END_IF;

      IF (*NOT algoritms.F2_Ch.autoAVOM_canrun_flag AND NOT algoritms.F2_R.autoAVOM_canrun_flag AND*) pnsoff.start THEN
  	    runPhase(Avom1Off);
  	    runPhase(Avom2Off);
  	    runPhase(Avom3Off);
  	    runPhase(Avom4Off);
  	    (*algoritms.R_AutoAVOM.CanRun:=FALSE;
  	    algoritms.R_AutoAVOM.reset();
  	    algoritms.S_AutoAVOM.CanRun:=FALSE;
  	    algoritms.S_AutoAVOM.reset();
  	    algoritms.Auto_Avom_.CanRun:=FALSE;*)
  	    runPhase(autoAVOMOff);
      END_IF;

      IF pnsOff.top AND Avom1Off.top AND Avom2Off.top AND Avom3Off.top AND Avom4Off.top AND autoAVOMOff.top  THEN
  	    runPhase(timer5);
      END_IF;

      IF timer5.top THEN
  	    runPhase(timer5);
      END_IF;
  END_IF;

  _sunpackerCommand(command := StrAlg.inCommand);
  	source := _sunpackerCommand.source;
  	cmd := _sunpackerCommand.cmd;

  IF cmd <> 0 AND lastCmd <> cmd AND (((NOT StrAlg.opcCommandsDisabled) AND source > 0) OR source = 0) then
  	CASE BYTE_TO_INT(cmd) OF
  		(*cmdRun*) 1: 	IF (StrAlg.CanRun) THEN
  					StrAlg.isRuning := TRUE;
  					StrAlg.isEnded := FALSE;
  					StrAlg.hasError := FALSE;
  					(*****************       OnRun       *****************)

                                                    algManager.nMode:=ModeGpa.MODE_NO;
                                                    (*runIfNotRunningSO(IM.SingleOutputs.Lampa_NO);*)

                                                    runPhase(kran4Close);
                                                    (*runPhase(timer120);*)
                                                    runPhase(nu1Off);
                                                    runPhase(timer600);

                                                   (* resetAiProtection(protections.Pgaza_na_vyhode_nagnetatelia);
                                                    resetAiProtection(protections.dPmaslo_gaz);
                                                    resetAiProtection(protections.Pmaslo_sm_nizkoe);
                                                    resetAiProtection(protections.Pmaslo_sm_vysokoe);
                                                    resetAiProtection(protections.Pgaza_na_vhode_nagnetatelia);
                                                    resetAiProtection(protections.Pgaza_na_vyhode_nagnetatelia);
                                                    resetDiProtection(protections.Reg_vozb_off);
                                                    resetDiProtection(protections.Fail_chastotnii_pusk);*)

  					cmd_for_Status := cmd;
  					source_for_Status := source;
  					command_error_for_Status := 0;
  				ELSE
  					StrAlg.isRuning := FALSE;
  					StrAlg.isEnded := FALSE;
  					StrAlg.hasError 	:= FALSE;

  					cmd_for_Status := 0;
  					source_for_Status := source;
  					command_error_for_Status := cmd;
  				END_IF;
  		(*cmdReset*) 2: 	StrAlg.isRuning := FALSE;
  				StrAlg.isEnded := FALSE;
  				StrAlg.hasError 	:= FALSE;

                                           (*****************       OnReset       *****************)
                                          waitReset(IN:=FALSE);
                                          (*resetIfRunningSO(IM.SingleOutputs.Lampa_NO);*)
                                          resetIfRunning(algoritms.vibegPNS);
                                          (*impulseSO(Im.SingleOutputs.SbrosBREO);*)

                                          (*resetPhase(timer120);*)
                                          resetPhase(kran6Open);
                                          resetPhase(pnsOn);
                                          resetPhase(kran4Close);
                                          resetPhase(kran3bOpen);
                                          resetPhase(mvOff);
                                          resetPhase(kran1Close);
                                          resetPhase(kran2Close);
                                          resetPhase(kran3Close);
                                          resetPhase(kran5Open);
  	                              (*resetPhase(error_Krans);*)
                                          resetPhase(autoPnsOff);
                                          resetPhase(pnsOn);
                                          resetPhase(Pg_VhodLessThen300);
                                          resetPhase(Pg_VyhodLessThen300);
                                          resetPhase(nu2Off);
                                          resetPhase(nu1Off);
                                          resetPhase(AutoNU_Off);
                                          resetPhase(timer600);

  				cmd_for_Status := cmd;
  				source_for_Status := source;
  				command_error_for_Status := 0;
  	END_CASE;
  	resetCmdTimer(IN := false);
  	resetCmdTimerPriznak := TRUE;
  END_IF;
  lastCmd := cmd;

  resetCmdTimer(IN := resetCmdTimerPriznak, PT := T#5S);
  IF resetCmdTimer.Q THEN
  	resetCmdTimerPriznak := FALSE;
  	source_for_Status := 0;
  	cmd_for_Status := 0;
  	command_error_for_Status := 0;
  END_IF;

  StrAlg.Start:= kran6Open.startStatus
              OR pnsOn.startStatus
              OR kran4Close.startStatus
              OR kran3bOpen.startStatus
              OR mvOff.startStatus
              OR kran1Close.startStatus
              OR kran2Close.startStatus
              OR kran3Close.startStatus
              OR kran5Open.startStatus
              OR Pg_VhodLessThen300.startStatus
              OR nu1off.startStatus
              OR nu2off.startStatus
              OR Pg_VyhodLessThen300.startStatus
              OR AutoNU_Off.startStatus
              OR timer600.startStatus
              OR pnsOff.startStatus
              OR Avom1Off.startStatus
              OR Avom2Off.startStatus
              OR Avom3Off.startStatus
              OR Avom4Off.startStatus
              OR autoAVOMOff.startStatus
              OR timer5.startStatus
              OR klapan1.startStatus
              OR klapan2.startStatus
              OR nu_On.startStatus
              OR Start_AO_From.startStatus;

  StrAlg.Error:= kran6Open.errorStatus
              OR pnsOn.errorStatus
              OR kran4Close.errorStatus
              OR kran3bOpen.errorStatus
              OR mvOff.errorStatus
              OR kran1Close.errorStatus
              OR kran2Close.errorStatus
              OR kran3Close.errorStatus
              OR kran5Open.errorStatus
              OR Pg_VhodLessThen300.errorStatus
              OR nu1off.errorStatus
              OR nu2off.errorStatus
              OR Pg_VyhodLessThen300.errorStatus
              OR AutoNU_Off.errorStatus
              OR timer600.errorStatus
              OR pnsOff.errorStatus
              OR Avom1Off.errorStatus
              OR Avom2Off.errorStatus
              OR Avom3Off.errorStatus
              OR Avom4Off.errorStatus
              OR autoAVOMOff.errorStatus
              OR timer5.errorStatus
              OR klapan1.errorStatus
              OR klapan2.errorStatus
              OR nu_On.errorStatus
              OR Start_AO_From.errorStatus;

  StrAlg.Top:= kran6Open.topStatus
              OR pnsOn.topStatus
              OR kran4Close.topStatus
              OR kran3bOpen.topStatus
              OR mvOff.topStatus
              OR kran1Close.topStatus
              OR kran2Close.topStatus
              OR kran3Close.topStatus
              OR kran5Open.topStatus
              OR Pg_VhodLessThen300.topStatus
              OR nu1off.topStatus
              OR nu2off.topStatus
              OR Pg_VyhodLessThen300.topStatus
              OR AutoNU_Off.topStatus
              OR timer600.topStatus
              OR pnsOff.topStatus
              OR Avom1Off.topStatus
              OR Avom2Off.topStatus
              OR Avom3Off.topStatus
              OR Avom4Off.topStatus
              OR autoAVOMOff.topStatus
              OR timer5.topStatus
              OR klapan1.topStatus
              OR klapan2.topStatus
              OR nu_On.topStatus
              OR Start_AO_From.topStatus;

  (*TODO: TYPE PROGRAM CODE HERE*)
  StrAlg.status :=  SHL(BYTE_TO_DWORD(source_for_Status), 29)
  			OR SHL(BYTE_TO_DWORD(cmd_for_Status), 26)
  			OR SHL(BYTE_TO_DWORD(command_error_for_Status), 23)
  			OR SHL(BOOL_TO_DWORD(StrAlg.OpcCommandsDisabled ), 21)
  			OR SHL(BOOL_TO_DWORD(StrAlg.hasError),4)
  			OR SHL(BOOL_TO_DWORD(StrAlg.CanRun),2)
  			OR SHL(BOOL_TO_DWORD(StrAlg.isEnded),1)
  			OR BOOL_TO_DWORD(StrAlg.isRuning);
END_FUNCTION_BLOCK

FUNCTION_BLOCK engineRunAlg
  VAR_IN_OUT
    StrAlg : struct_Alg;
  END_VAR
  VAR
    BreakPuskTimer : struct_PhaseAlgoritm;
    RunProtection_mvoff : struct_PhaseAlgoritm;
    LowOil_upStopust : struct_PhaseAlgoritm;
    mvOn : struct_PhaseAlgoritm;
    AutoPns_ph : struct_PhaseAlgoritm;
    AutoAvom_ph : struct_PhaseAlgoritm;
    pnsOff : struct_PhaseAlgoritm;
    testUnsuccessful : struct_PhaseAlgoritm;
    fb_BreakPuskTimer : fb_ph_Timer;
    fb_RunProtection_mvoff : fb_ph_DIprotection;
    fb_LowOil_upStopust : fb_ph_WaitAnalogValue;
    fb_mvOn : fb_ph_SectionSwitch;
    fb_AutoPns_ph : fb_ph_algoritm;
    fb_AutoAvom_ph : fb_ph_algoritm;
    fb_pnsOff : fb_ph_Switch;
    fb_testUnsuccessful : fb_ph_CustomPhase;
    _sunpackerCommand : fb_sunpackerCommand;
    _DualStateImAction : TYPE_DualStateImAction;
    _PhaseAlgoritmAction : TYPE_PhaseAlgoritmAction;
    source : BYTE;
    cmd : BYTE;
    lastCmd : BYTE;
    source_for_Status : BYTE;
    cmd_for_Status : BYTE;
    command_error_for_Status : BYTE;
    resetCmdTimer : TON;
    resetCmdTimerPriznak : BOOL;
    onInit : BOOL;
    waitReset : TON;
  END_VAR
  VAR_EXTERNAL
    IM : ImConfig;
    algoritms : AlgoritmsConfig;
    ai : AiConfig;
    protections : ProtectionsConfig;
    AlgTimers : struct_AlgTimers;
  END_VAR

  IF NOT onInit THEN

       fb_BreakPuskTimer(phaseNumber:=0, delay:=T#665S);
     fb_LowOil_upStopust(phaseNumber:=1);
                 fb_mvOn(phaseNumber:=2, act:=_on);
           fb_AutoPns_ph(phaseNumber:=3, act:=_run, waitCompletion:=FALSE);
          fb_AutoAvom_ph(phaseNumber:=4, act:=_run, waitCompletion:=FALSE);
               fb_pnsOff(phaseNumber:=5, act:=_off);
  fb_RunProtection_mvoff(phaseNumber:=7, act:=_run);
     fb_testUnsuccessful(phaseNumber:=17);

  onInit:=TRUE;
  END_IF;

          fb_BreakPuskTimer(StrPh:=BreakPuskTimer, timer:=AlgTimers.engineRun_BreakPuskTimer);
       (* fb_LowOil_upStopust(StrPh:=LowOil_upStopust, ai:=ai.Pmasla_posle_GNS, more:=im.AutoPns_UstStop.Value);*)
                    fb_mvOn(StrPh:=mvOn, Im:=Im.mv);
              fb_AutoPns_ph(StrPh:=AutoPns_ph, alg:=algoritms.AutoPns);
             fb_AutoAvom_ph(StrPh:=AutoAvom_ph, alg:=algoritms.AutoAvom);
                  fb_pnsOff(StrPh:=pnsOff, Im:=Im.pns);
    (*fb_RunProtection_mvoff(StrPh:=RunProtection_mvoff, StrDiP:=protections.Pgaza_na_vyhode_nagnetatelia_GPA_STOP);*)
        fb_testUnsuccessful(StrPh:=testUnsuccessful);

  StrAlg.CanRun := StrAlg.inCanRun;
  StrAlg.OpcCommandsDisabled := StrAlg.inOpcCommandsDisabled;

  IF StrAlg.isRuning THEN

      StrAlg.hasError := mvOn.error OR pnsOff.error OR testUnsuccessful.error;

      IF mvOn.top THEN
          runPhase(RunProtection_mvoff);
          runPhase(AutoAvom_ph);
          runPhase(LowOil_upStopust);
      END_IF;
      (*
      IF AutoAvom_ph.top THEN
          algoritms.AutoAvom.inOpcCommandsDisabled:=FALSE;
      END_IF;
      *)
      IF LowOil_upStopust.top THEN
          runPhase(pnsOff);
      END_IF;

      IF pnsOff.top THEN
         runPhase(AutoPns_ph);
      END_IF;

      IF BreakPuskTimer.top AND NOT AutoPns_ph.top THEN
            testUnsuccessful.error:=TRUE;
      END_IF;

      IF AutoPns_ph.top THEN
            resetPhase(BreakPuskTimer);
  	waitReset(IN:=TRUE, PT:= T#2S);
      END_IF;

      IF waitReset.Q AND NOT (algoritms.Apusk.isRuning OR algoritms.SemiAutoPusk.isRuning) THEN
  	resetIfRunning(StrAlg);
      END_IF;

      StrAlg.isEnded:= AutoPns_ph.top;
  END_IF;

  StrAlg.CanRun := StrAlg.inCanRun;
  StrAlg.OpcCommandsDisabled := StrAlg.inOpcCommandsDisabled;

  (* ---- Если управление с ВУ заблокировано, то  передаем команду из алгоритма ---- *)
  IF StrAlg.inOpcCommandsDisabled THEN
  	StrAlg.inCommand := StrAlg.inCommand_Alg;
  ELSE (* иначе передаем команду с АРМа*)
  	StrAlg.inCommand := StrAlg.inCommand_ARM;
  END_IF;

  _sunpackerCommand(command := StrAlg.inCommand);
  	source := _sunpackerCommand.source;
  	cmd := _sunpackerCommand.cmd;

  IF cmd <> 0 AND lastCmd <> cmd AND (((NOT StrAlg.opcCommandsDisabled) AND source > 0) OR source = 0) then
  	CASE BYTE_TO_INT(cmd) OF
  		(*cmdRun*) 1: 	IF (StrAlg.CanRun) THEN
  					StrAlg.isRuning := TRUE;
  					StrAlg.isEnded := FALSE;
  					StrAlg.hasError := FALSE;
  					(*****************       OnRun       *****************)

                                                    runPhase(mvOn);
                                                    runPhase(BreakPuskTimer);
                                                    runPhase(testUnsuccessful);

  					cmd_for_Status := cmd;
  					source_for_Status := source;
  					command_error_for_Status := 0;
  				ELSE
  					StrAlg.isRuning := FALSE;
  					StrAlg.isEnded := FALSE;
  					StrAlg.hasError 	:= FALSE;

  					cmd_for_Status := 0;
  					source_for_Status := source;
  					command_error_for_Status := cmd;
  				END_IF;
  		(*cmdReset*) 2: 	StrAlg.isRuning := FALSE;
  				StrAlg.isEnded := FALSE;
  				StrAlg.hasError 	:= FALSE;

                                           (*****************       OnReset       *****************)
                                          StrAlg.inCanRun:=FALSE;
                                          waitReset(IN:=FALSE);

                                          resetPhase(BreakPuskTimer);
                                          resetPhase(RunProtection_mvoff);
                                          resetPhase(LowOil_upStopust);
                                          resetPhase(mvOn);
                                          resetPhase(AutoPns_ph);
                                          resetPhase(AutoAvom_ph);
                                          resetPhase(pnsOff);
                                          resetPhase(testUnsuccessful);

  				cmd_for_Status := cmd;
  				source_for_Status := source;
  				command_error_for_Status := 0;
  	END_CASE;
  	resetCmdTimer(IN := false);
  	resetCmdTimerPriznak := TRUE;
  END_IF;
  lastCmd := cmd;

  resetCmdTimer(IN := resetCmdTimerPriznak, PT := T#5S);
  IF resetCmdTimer.Q THEN
  	resetCmdTimerPriznak := FALSE;
  	source_for_Status := 0;
  	cmd_for_Status := 0;
  	command_error_for_Status := 0;
  END_IF;

  StrAlg.Start:= BreakPuskTimer.startStatus
              OR RunProtection_mvoff.startStatus
              OR LowOil_upStopust.startStatus
              OR mvOn.startStatus
              OR AutoPns_ph.startStatus
              OR AutoAvom_ph.startStatus
              OR pnsOff.startStatus
              OR testUnsuccessful.startStatus;

  StrAlg.Error:= BreakPuskTimer.errorStatus
              OR RunProtection_mvoff.errorStatus
              OR LowOil_upStopust.errorStatus
              OR mvOn.errorStatus
              OR AutoPns_ph.errorStatus
              OR AutoAvom_ph.errorStatus
              OR pnsOff.errorStatus
              OR testUnsuccessful.errorStatus;

  StrAlg.Top:=   BreakPuskTimer.topStatus
              OR RunProtection_mvoff.topStatus
              OR LowOil_upStopust.topStatus
              OR mvOn.topStatus
              OR AutoPns_ph.topStatus
              OR AutoAvom_ph.topStatus
              OR pnsOff.topStatus
              OR testUnsuccessful.topStatus;

  (*TODO: TYPE PROGRAM CODE HERE*)
  StrAlg.status :=  SHL(BYTE_TO_DWORD(source_for_Status), 29)
  			OR SHL(BYTE_TO_DWORD(cmd_for_Status), 26)
  			OR SHL(BYTE_TO_DWORD(command_error_for_Status), 23)
  			OR SHL(BOOL_TO_DWORD(StrAlg.OpcCommandsDisabled ), 21)
  			OR SHL(BOOL_TO_DWORD(StrAlg.hasError),4)
  			OR SHL(BOOL_TO_DWORD(StrAlg.CanRun),2)
  			OR SHL(BOOL_TO_DWORD(StrAlg.isEnded),1)
  			OR BOOL_TO_DWORD(StrAlg.isRuning);
END_FUNCTION_BLOCK

FUNCTION_BLOCK puskKalg
  VAR_IN_OUT
    StrAlg : struct_Alg;
  END_VAR
  VAR
    puskOilSystem : struct_PhaseAlgoritm;
  END_VAR
  VAR_IN_OUT
    questionFilling : struct_Question;
  END_VAR
  VAR
    filling : struct_PhaseAlgoritm;
  END_VAR
  VAR_IN_OUT
    questionUnload : struct_Question;
  END_VAR
  VAR
    kran3bOpen : struct_PhaseAlgoritm;
    kran4Close : struct_PhaseAlgoritm;
    kran1Close : struct_PhaseAlgoritm;
    kran2Close : struct_PhaseAlgoritm;
    kran5open : struct_PhaseAlgoritm;
    wait720 : struct_PhaseAlgoritm;
    noGasInPipe : struct_PhaseAlgoritm;
    AutoNUoff : struct_PhaseAlgoritm;
    nu1Off : struct_PhaseAlgoritm;
    nu2Off : struct_PhaseAlgoritm;
    pnsWaitOff : struct_PhaseAlgoritm;
    testUnsuccessfulUnfill : struct_PhaseAlgoritm;
    fb_puskOilSystem : fb_ph_algoritm;
    fb_questionFilling : fb_Question;
    fb_filling : fb_ph_algoritm;
    fb_questionUnload : fb_Question;
    fb_kran3bOpen : fb_ph_Kran;
    fb_kran4Close : fb_ph_CustomPhase;
    fb_kran1Close : fb_ph_Kran;
    fb_kran2Close : fb_ph_Kran;
    fb_kran5open : fb_ph_Kran;
    fb_wait720 : fb_ph_Timer;
    fb_noGasInPipe : fb_ph_CustomPhase;
    fb_AutoNUoff : fb_ph_algoritm;
    fb_nu1Off : fb_ph_OilPump;
    fb_nu2Off : fb_ph_OilPump;
    fb_pnsWaitOff : fb_ph_algoritm;
    fb_testUnsuccessfulUnfill : fb_ph_CustomPhase;
    _sunpackerCommand : fb_sunpackerCommand;
    _DualStateImAction : TYPE_DualStateImAction;
    _Answers : TYPE_Answers;
    _statusDualInput : TYPE_statusDualInput;
    _StatusAi : TYPE_StatusAi;
    _PhaseAlgoritmAction : TYPE_PhaseAlgoritmAction;
    source : BYTE;
    cmd : BYTE;
    lastCmd : BYTE;
    source_for_Status : BYTE;
    cmd_for_Status : BYTE;
    command_error_for_Status : BYTE;
    resetCmdTimer : TON;
    resetCmdTimerPriznak : BOOL;
    OpcCommandsKransEnabled : BOOL;
    OpcCommandsKransDisabled : BOOL;
    _resetQuestion1 : BOOL;
    _resetQuestion2 : BOOL;
    onInit : BOOL;
    waitReset : TON;
  END_VAR
  VAR_EXTERNAL
    IM : ImConfig;
    algoritms : AlgoritmsConfig;
    ai : AiConfig;
    AlgTimers : struct_AlgTimers;
    ModeGpa : TYPE_ModeGpa;
    algManager : struct_AlgoritmsManager;
    protections : ProtectionsConfig;
  END_VAR
  VAR CONSTANT
    Ust_Pgaza : LREAL          := 0.3;
  END_VAR

  IF NOT onInit THEN

            fb_puskOilSystem(phaseNumber:=0, act:=_run, waitCompletion:=TRUE);
        questionFilling.AnswerVariants:=_Answers.ANS_YES;
                  fb_filling(phaseNumber:=1, act:=_run, waitCompletion:=TRUE);
      questionUnload.AnswerVariants:=_Answers.ANS_YES;
               fb_kran3bOpen(phaseNumber:=3, act:=_on);
               fb_kran4Close(phaseNumber:=4);
               fb_kran1Close(phaseNumber:=5, act:=_off);
               fb_kran2Close(phaseNumber:=6, act:=_off);
                fb_kran5open(phaseNumber:=7, act:=_on);
                  fb_wait720(phaseNumber:=8, delay:=T#720S);
              fb_noGasInPipe(phaseNumber:=9);
                fb_AutoNUoff(phaseNumber:=10, act:=_reset, waitCompletion:=FALSE);
                   fb_nu1Off(phaseNumber:=11, act:=_off);
                   fb_nu2Off(phaseNumber:=12, act:=_off);
               fb_pnsWaitOff(phaseNumber:=15, act:=_run, waitCompletion:=TRUE);
   fb_testUnsuccessfulUnfill(phaseNumber:=18);

  onInit:=TRUE;
  END_IF;

            fb_puskOilSystem(StrPh:=puskOilSystem, alg:=algoritms.puskOilSystem);
          fb_questionFilling(StrQ:=questionFilling);
                  fb_filling(StrPh:=filling, alg:=algoritms.filling);
           fb_questionUnload(StrQ:=questionUnload);
               fb_kran3bOpen(StrPh:=kran3bOpen, Im:=Im.kran3b);
               fb_kran4Close(StrPh:=kran4Close);
               fb_kran1Close(StrPh:=kran1Close, Im:=Im.kran1);
               fb_kran2Close(StrPh:=kran2Close, Im:=Im.kran2);
                fb_kran5open(StrPh:=kran5open, Im:=Im.kran5);
                  fb_wait720(StrPh:=wait720, timer:=AlgTimers.puskK_wait720);
              fb_noGasInPipe(StrPh:=noGasInPipe);
                fb_AutoNUoff(StrPh:=AutoNUoff, alg:=algoritms.autoNu);
                   fb_nu1Off(StrPh:=nu1Off, Im:=Im.nu1);
                   fb_nu2Off(StrPh:=nu2Off, Im:=Im.nu2);
               fb_pnsWaitOff(StrPh:=pnsWaitOff, alg:=algoritms.vibegPNS);
   fb_testUnsuccessfulUnfill(StrPh:=testUnsuccessfulUnfill);

  StrAlg.CanRun := StrAlg.inCanRun;
  StrAlg.OpcCommandsDisabled := StrAlg.inOpcCommandsDisabled;

  IF StrAlg.isRuning THEN

      StrAlg.hasError := kran3bOpen.error OR kran1Close.error OR kran2Close.error OR kran5open.error OR testUnsuccessfulUnfill.error;

      IF puskOilSystem.top THEN
           IF NOT _resetQuestion1 THEN
           askQuestion(questionFilling);
           _resetQuestion1:=TRUE;
           END_IF;
      END_IF;

      IF questionFilling.answer = _Answers.ANS_YES THEN
          runPhase(filling);
          resetQuestion(questionFilling);
      END_IF;

      IF filling.top THEN
         OpcCommandsKransEnabled:=TRUE;
         resetDiProtection(protections.Reg_vozb_off);
         (*resetDiProtection(protections.Fail_chastotnii_pusk);*)
         IF NOT _resetQuestion2 THEN
         askQuestion(questionUnload);
         _resetQuestion2:=TRUE;
         END_IF;
      END_IF;

       IF questionUnload.answer = _Answers.ANS_YES THEN
          OpcCommandsKransDisabled:=TRUE;
          runPhase(kran3bOpen);
          runPhase(wait720);
          resetQuestion(questionUnload);
      END_IF;

      IF kran3bOpen.top THEN
            resetDiProtection(protections.Reg_vozb_off);
            resetDiProtection(protections.Fail_chastotnii_pusk);

            runPhase(kran1Close);
            runPhase(kran2Close);
            runPhase(kran4Close);
      END_IF;

       IF kran4Close.start AND NOT kran4Close.top THEN
  	kran4Close.top:= Im.kran4.onStatus = _statusDualInput.STATUS_OFF;
      END_IF;

      IF kran1Close.top AND kran2Close.top AND kran4Close.top THEN
  	runPhase(kran5open);
      END_IF;

      IF kran5open.top THEN
  	runPhase(noGasInPipe);
      END_IF;

      IF noGasInPipe.start AND (NOT noGasInPipe.top) THEN
  	noGasInPipe.top:=  (ai.dPgaza_na_maslo_filtre.interval >= _statusAi.NORMAL
                           AND  ai.dPgaza_na_maslo_filtre.value< Ust_Pgaza )
                           AND (ai.Pmaslo_sm_vysokoe.interval >= _statusAi.NORMAL
                           AND  ai.Pmaslo_sm_vysokoe.value< Ust_Pgaza);
      END_IF;

      IF noGasInPipe.top THEN

            ai.Tmasla_MB.Disabled_LA:=TRUE;
            ai.Tmasla_MB.Disabled_LW:=TRUE;
            (*IM.SingleSignals.dP_oilgaz_low.Disabled_Sig:=TRUE;*)
            resetAiProtection(protections.Os_sdvig_nagnetatelja_plus);
           (* resetDiProtection(protections.Vibro_skorost_OP_shesterni_RED_T5);*)
  	runPhase(AutoNUoff);

      END_IF;

       IF autoNuOff.top THEN
  	runPhase(nu1off);
            runPhase(nu2off);
      END_IF;

      IF nu1Off.top AND nu2Off.top THEN
  	runPhase(pnsWaitOff);
      END_IF;

      IF wait720.top AND NOT (pnsWaitOff.top) THEN
            testUnsuccessfulUnfill.error:=TRUE;
      END_IF;

      IF pnsWaitOff.top THEN
            resetPhase(wait720);
  	waitReset(IN:=TRUE, PT:= T#3S);
      END_IF;

      IF waitReset.Q THEN
          resetIfRunning(algoritms.vibegPNS);
          algManager.nMode:=ModeGpa.MODE_STOP;
          resetIfRunning(StrAlg);
      END_IF;

      StrAlg.isEnded:= pnsWaitOff.top;

      IF OpcCommandsKransEnabled AND NOT OpcCommandsKransDisabled THEN
  	IF      (im.pns.onStatus = _statusDualInput.STATUS_ON)
                AND (im.nu1.onStatus = _statusDualInput.STATUS_ON OR im.nu2.onStatus = _statusDualInput.STATUS_ON)
  	    AND (ai.Tmasla_MB.interval >= _statusAi.normal)
                (*AND (ai.Tmasla_MB.value > im.PuskOilSystem_UstdPmg.Value)*)
            THEN
  	    IM.Kran3b.inOpcCommandsDisabled:=FALSE;
  	    Im.kran4.inOpcCommandsDisabled:=FALSE;
  	    Im.kran5.inOpcCommandsDisabled:=FALSE;
  		(*IF	Im.SingleSignals.dP_gazgaz_Kran1.q THEN
  			Im.kran1.inOpcCommandsDisabled:=FALSE;
  			Im.kran2.inOpcCommandsDisabled:=FALSE;
  		ELSE
  			Im.kran1.inOpcCommandsDisabled:=TRUE;
  			Im.kran2.inOpcCommandsDisabled:=TRUE;
  		END_IF;*)
            ELSE
  	    Im.kran1.inOpcCommandsDisabled:=TRUE;
  	    Im.kran2.inOpcCommandsDisabled:=TRUE;
  	    Im.kran3b.inOpcCommandsDisabled:=TRUE;
  	    Im.kran4.inOpcCommandsDisabled:=TRUE;
  	    Im.kran5.inOpcCommandsDisabled:=TRUE;
            END_IF;

      ELSE
  	Im.kran1.inOpcCommandsDisabled:=TRUE;
  	Im.kran2.inOpcCommandsDisabled:=TRUE;
  	Im.kran3b.inOpcCommandsDisabled:=TRUE;
  	Im.kran4.inOpcCommandsDisabled:=TRUE;
  	Im.kran5.inOpcCommandsDisabled:=TRUE;
      END_IF;
  END_IF;

  StrAlg.CanRun := StrAlg.inCanRun;
  StrAlg.OpcCommandsDisabled := StrAlg.inOpcCommandsDisabled;

  (* ---- Если управление с ВУ заблокировано, то  передаем команду из алгоритма ---- *)
  IF StrAlg.inOpcCommandsDisabled THEN
  	StrAlg.inCommand := StrAlg.inCommand_Alg;
  ELSE (* иначе передаем команду с АРМа*)
  	StrAlg.inCommand := StrAlg.inCommand_ARM;
  END_IF;

  _sunpackerCommand(command := StrAlg.inCommand);
  	source := _sunpackerCommand.source;
  	cmd := _sunpackerCommand.cmd;

  IF cmd <> 0 AND lastCmd <> cmd AND (((NOT StrAlg.opcCommandsDisabled) AND source > 0) OR source = 0) then
  	CASE BYTE_TO_INT(cmd) OF
  		(*cmdRun*) 1: 	IF (StrAlg.CanRun) THEN
  					StrAlg.isRuning := TRUE;
  					StrAlg.isEnded := FALSE;
  					StrAlg.hasError := FALSE;
  					(*****************       OnRun       *****************)

                                                    algManager.nMode:=ModeGpa.MODE_PUSKK;
                                                    resetAndDisable(alg:=algoritms.ppu);
                                                    algoritms.puskOilSystem.inCanRun:= TRUE;
                                                    algoritms.filling.inCanRun:= TRUE;
                                                    runPhase(puskOilSystem);

  					cmd_for_Status := cmd;
  					source_for_Status := source;
  					command_error_for_Status := 0;
  				ELSE
  					StrAlg.isRuning := FALSE;
  					StrAlg.isEnded := FALSE;
  					StrAlg.hasError 	:= FALSE;

  					cmd_for_Status := 0;
  					source_for_Status := source;
  					command_error_for_Status := cmd;
  				END_IF;
  		(*cmdReset*) 2: 	StrAlg.isRuning := FALSE;
  				StrAlg.isEnded := FALSE;
  				StrAlg.hasError 	:= FALSE;

                                           (*****************       OnReset       *****************)
                                          OpcCommandsKransEnabled:=FALSE;
                                          OpcCommandsKransDisabled:=FALSE;
                                          waitReset(IN:=FALSE);
                                          _resetQuestion1:=FALSE;
                                          _resetQuestion2:=FALSE;
                                          resetPhase(puskOilSystem);
                                          resetPhase(filling);
                                          resetPhase(kran3bOpen);
                                          resetPhase(kran4Close);
                                          resetPhase(kran1Close);
                                          resetPhase(kran2Close);
                                          resetPhase(kran5open);
                                          resetPhase(wait720);
                                          resetPhase(noGasInPipe);
                                          resetPhase(AutoNUoff);
                                          resetPhase(nu1Off);
                                          resetPhase(nu2Off);
                                          resetPhase(pnsWaitOff);
                                          resetPhase(testUnsuccessfulUnfill);
                                          BlockAllIM(IM);
                                          resetQuestion(questionFilling);
                                          resetQuestion(questionUnload);

                                          StrAlg.inOpcCommandsDisabled:=FALSE;

  				cmd_for_Status := cmd;
  				source_for_Status := source;
  				command_error_for_Status := 0;
  	END_CASE;
  	resetCmdTimer(IN := false);
  	resetCmdTimerPriznak := TRUE;
  END_IF;
  lastCmd := cmd;

  resetCmdTimer(IN := resetCmdTimerPriznak, PT := T#5S);
  IF resetCmdTimer.Q THEN
  	resetCmdTimerPriznak := FALSE;
  	source_for_Status := 0;
  	cmd_for_Status := 0;
  	command_error_for_Status := 0;
  END_IF;

  StrAlg.Start:= puskOilSystem.startStatus
              OR filling.startStatus
              OR kran3bOpen.startStatus
              OR kran4Close.startStatus
              OR kran1Close.startStatus
              OR kran2Close.startStatus
              OR kran5open.startStatus
              OR wait720.startStatus
              OR noGasInPipe.startStatus
              OR AutoNUoff.startStatus
              OR nu1Off.startStatus
              OR nu2Off.startStatus
              OR pnsWaitOff.startStatus
              OR testUnsuccessfulUnfill.startStatus;

  StrAlg.Error:=  puskOilSystem.errorStatus
              OR filling.errorStatus
              OR kran3bOpen.errorStatus
              OR kran4Close.errorStatus
              OR kran1Close.errorStatus
              OR kran2Close.errorStatus
              OR kran5open.errorStatus
              OR wait720.errorStatus
              OR noGasInPipe.errorStatus
              OR AutoNUoff.errorStatus
              OR nu1Off.errorStatus
              OR nu2Off.errorStatus
              OR pnsWaitOff.errorStatus
              OR testUnsuccessfulUnfill.errorStatus;

  StrAlg.Top:=   puskOilSystem.topStatus
              OR filling.topStatus
              OR kran3bOpen.topStatus
              OR kran4Close.topStatus
              OR kran1Close.topStatus
              OR kran2Close.topStatus
              OR kran5open.topStatus
              OR wait720.topStatus
              OR noGasInPipe.topStatus
              OR AutoNUoff.topStatus
              OR nu1Off.topStatus
              OR nu2Off.topStatus
              OR pnsWaitOff.topStatus
              OR testUnsuccessfulUnfill.topStatus;

  (*TODO: TYPE PROGRAM CODE HERE*)
  StrAlg.status :=  SHL(BYTE_TO_DWORD(source_for_Status), 29)
  			OR SHL(BYTE_TO_DWORD(cmd_for_Status), 26)
  			OR SHL(BYTE_TO_DWORD(command_error_for_Status), 23)
  			OR SHL(BOOL_TO_DWORD(StrAlg.OpcCommandsDisabled ), 21)
  			OR SHL(BOOL_TO_DWORD(StrAlg.hasError),4)
  			OR SHL(BOOL_TO_DWORD(StrAlg.CanRun),2)
  			OR SHL(BOOL_TO_DWORD(StrAlg.isEnded),1)
  			OR BOOL_TO_DWORD(StrAlg.isRuning);
END_FUNCTION_BLOCK

FUNCTION_BLOCK puskValg
  VAR_IN_OUT
    StrAlg : struct_Alg;
  END_VAR
  VAR
    puskOilSystem : struct_PhaseAlgoritm;
  END_VAR
  VAR_IN_OUT
    questionEngine : struct_Question;
  END_VAR
  VAR
    runningEngine : struct_PhaseAlgoritm;
  END_VAR
  VAR_IN_OUT
    questionMVoff : struct_Question;
  END_VAR
  VAR
    mvOff : struct_PhaseAlgoritm;
    pnsOn : struct_PhaseAlgoritm;
    wait600 : struct_PhaseAlgoritm;
    AutoNUoff : struct_PhaseAlgoritm;
    nu1Off : struct_PhaseAlgoritm;
    nu2Off : struct_PhaseAlgoritm;
    autoAvomOff : struct_PhaseAlgoritm;
    Avom1Off : struct_PhaseAlgoritm;
    Avom2Off : struct_PhaseAlgoritm;
    pnsWaitOff : struct_PhaseAlgoritm;
    testUnsuccessful : struct_PhaseAlgoritm;
    fb_puskOilSystem : fb_ph_algoritm;
    fb_questionEngine : fb_Question;
    fb_runningEngine : fb_ph_algoritm;
    fb_questionMVoff : fb_Question;
    fb_mvOff : fb_ph_SectionSwitch;
    fb_pnsOn : fb_ph_Switch;
    fb_wait600 : fb_ph_Timer;
    fb_AutoNUoff : fb_ph_algoritm;
    fb_nu1Off : fb_ph_OilPump;
    fb_nu2Off : fb_ph_OilPump;
    fb_autoAvomOff : fb_ph_algoritm;
    fb_Avom1Off : fb_ph_Switch;
    fb_Avom2Off : fb_ph_Switch;
    fb_pnsWaitOff : fb_ph_algoritm;
    fb_testUnsuccessful : fb_ph_CustomPhase;
    _sunpackerCommand : fb_sunpackerCommand;
    _DualStateImAction : TYPE_DualStateImAction;
    _Answers : TYPE_Answers;
    _statusDualInput : TYPE_statusDualInput;
    _StatusAi : TYPE_StatusAi;
    _PhaseAlgoritmAction : TYPE_PhaseAlgoritmAction;
    source : BYTE;
    cmd : BYTE;
    lastCmd : BYTE;
    source_for_Status : BYTE;
    cmd_for_Status : BYTE;
    command_error_for_Status : BYTE;
    resetCmdTimer : TON;
    resetCmdTimerPriznak : BOOL;
    onInit : BOOL;
    _resetQuestion1 : BOOL;
    _resetQuestion2 : BOOL;
    waitReset : TON;
  END_VAR
  VAR_EXTERNAL
    IM : ImConfig;
    algoritms : AlgoritmsConfig;
    ai : AiConfig;
    AlgTimers : struct_AlgTimers;
    ModeGpa : TYPE_ModeGpa;
    algManager : struct_AlgoritmsManager;
    protections : ProtectionsConfig;
  END_VAR
  VAR CONSTANT
    Ust_Pgaza : LREAL          := 0.3;
  END_VAR

  IF NOT onInit THEN

            fb_puskOilSystem(phaseNumber:=0, act:=_run, waitCompletion:=TRUE);
         questionEngine.AnswerVariants:=_Answers.ANS_YES;
            fb_runningEngine(phaseNumber:=1, act:=_run, waitCompletion:=TRUE);
          questionMVoff.AnswerVariants:=_Answers.ANS_YES;
                    fb_mvOff(phaseNumber:=3, act:=_off);
                    fb_pnsOn(phaseNumber:=4, act:=_on);
                  fb_wait600(phaseNumber:=8, delay:=T#600S);
                fb_AutoNUoff(phaseNumber:=10, act:=_reset, waitCompletion:=FALSE);
                   fb_nu1Off(phaseNumber:=11, act:=_off);
                   fb_nu2Off(phaseNumber:=12, act:=_off);
               fb_pnsWaitOff(phaseNumber:=15, act:=_run, waitCompletion:=TRUE);
              fb_autoAvomOff(phaseNumber:=7, act:=_reset, waitCompletion:=FALSE);
                 fb_Avom1Off(phaseNumber:=5, act:=_off);
                 fb_Avom2Off(phaseNumber:=6, act:=_off);
         fb_testUnsuccessful(phaseNumber:=17);

  onInit:=TRUE;
  END_IF;

            fb_puskOilSystem(StrPh:=puskOilSystem, alg:=algoritms.puskOilSystem);
           fb_questionEngine(StrQ:=questionEngine);
            fb_runningEngine(StrPh:=runningEngine, alg:=algoritms.engineRun);
            fb_questionMVoff(StrQ:=questionMVoff);
                    fb_mvOff(StrPh:=mvOff, Im:=Im.mv);
                    fb_pnsOn(StrPh:=pnsOn, Im:=Im.pns);
                  fb_wait600(StrPh:=wait600, timer:=AlgTimers.puskV_wait600);
                fb_AutoNUoff(StrPh:=AutoNUoff, alg:=algoritms.autoNu);
                   fb_nu1Off(StrPh:=nu1Off, Im:=Im.nu1);
                   fb_nu2Off(StrPh:=nu2Off, Im:=Im.nu2);
               fb_pnsWaitOff(StrPh:=pnsWaitOff, alg:=algoritms.vibegPNS);
              fb_autoAvomOff(StrPh:=autoAvomOff, alg:=algoritms.AutoAvom);
                 fb_Avom1Off(StrPh:=Avom1Off, Im:=Im.v1_Avom);
                 fb_Avom2Off(StrPh:=Avom2Off, Im:=Im.v2_Avom);
         fb_testUnsuccessful(StrPh:=testUnsuccessful);

  StrAlg.CanRun := StrAlg.inCanRun;
  StrAlg.OpcCommandsDisabled := StrAlg.inOpcCommandsDisabled;

  IF StrAlg.isRuning THEN

      StrAlg.hasError := mvOff.error OR pnsOn.error OR testUnsuccessful.error;

      IF puskOilSystem.top THEN
           IF NOT _resetQuestion1 THEN
           askQuestion(questionEngine);
           _resetQuestion1:=TRUE;
           END_IF;
      END_IF;

      IF questionEngine.answer = _Answers.ANS_YES THEN
          runPhase(runningEngine);
          resetQuestion(questionEngine);
      END_IF;

      IF runningEngine.top THEN
         IF NOT _resetQuestion2 THEN
         askQuestion(questionMVoff);
         _resetQuestion2:=TRUE;
         END_IF;
      END_IF;

       IF questionMVoff.answer = _Answers.ANS_YES THEN

          (*resetDiProtection(protections.Pgaza_na_vyhode_nagnetatelia_GPA_STOP);
         *) resetIfRunning(algoritms.AutoPns);
          runPhase(mvOff);
          runPhase(wait600);
          resetQuestion(questionMVoff);
       END_IF;

      IF mvOff.top THEN
          runPhase(pnsOn);
      END_IF;

      IF pnsOn.top THEN

            ai.Tmasla_MB.Disabled_LA:=TRUE;
            ai.Tmasla_MB.Disabled_LW:=TRUE;
            (*IM.SingleSignals.dP_oilgaz_low.Disabled_Sig:=TRUE;*)
            (*resetAiProtection(protections.Os_sdvig_nagnetatelja_plus)*)
           (* resetDiProtection(protections.Vibro_skorost_OP_shesterni_RED_T5);*)
  	runPhase(AutoNUoff);

      END_IF;

       IF autoNuOff.top THEN
  	runPhase(nu1off);
            runPhase(nu2off);
      END_IF;

      IF nu1Off.top AND nu2Off.top THEN
  	runPhase(pnsWaitOff);
      END_IF;

      IF wait600.top AND NOT (pnsWaitOff.top) THEN
            testUnsuccessful.error:=TRUE;
      END_IF;

      IF pnsWaitOff.top THEN
            resetPhase(wait600);
            runPhase(autoAvomOff);
  	waitReset(IN:=TRUE, PT:= T#3S);
      END_IF;

      IF autoAvomOff.top THEN
            runPhase(Avom1Off);
            runPhase(Avom2Off);
      END_IF;

      IF waitReset.Q THEN
          resetIfRunning(algoritms.vibegPNS);
          algManager.nMode:=ModeGpa.MODE_STOP;
          resetIfRunning(StrAlg);
      END_IF;

      StrAlg.isEnded:= pnsWaitOff.top;

  END_IF;

  StrAlg.CanRun := StrAlg.inCanRun;
  StrAlg.OpcCommandsDisabled := StrAlg.inOpcCommandsDisabled;

  (* ---- Если управление с ВУ заблокировано, то  передаем команду из алгоритма ---- *)
  IF StrAlg.inOpcCommandsDisabled THEN
  	StrAlg.inCommand := StrAlg.inCommand_Alg;
  ELSE (* иначе передаем команду с АРМа*)
  	StrAlg.inCommand := StrAlg.inCommand_ARM;
  END_IF;

  _sunpackerCommand(command := StrAlg.inCommand);
  	source := _sunpackerCommand.source;
  	cmd := _sunpackerCommand.cmd;

  IF cmd <> 0 AND lastCmd <> cmd AND (((NOT StrAlg.opcCommandsDisabled) AND source > 0) OR source = 0) then
  	CASE BYTE_TO_INT(cmd) OF
  		(*cmdRun*) 1: 	IF (StrAlg.CanRun) THEN
  					StrAlg.isRuning := TRUE;
  					StrAlg.isEnded := FALSE;
  					StrAlg.hasError := FALSE;
  					(*****************       OnRun       *****************)

                                                    algManager.nMode:=ModeGpa.MODE_PUSKV;
                                                    resetAndDisable(alg:=algoritms.ppu);
                                                    algoritms.puskOilSystem.inCanRun:= TRUE;
                                                    algoritms.engineRun.inCanRun:= TRUE;
                                                    runPhase(puskOilSystem);

  					cmd_for_Status := cmd;
  					source_for_Status := source;
  					command_error_for_Status := 0;
  				ELSE
  					StrAlg.isRuning := FALSE;
  					StrAlg.isEnded := FALSE;
  					StrAlg.hasError 	:= FALSE;

  					cmd_for_Status := 0;
  					source_for_Status := source;
  					command_error_for_Status := cmd;
  				END_IF;
  		(*cmdReset*) 2: 	StrAlg.isRuning := FALSE;
  				StrAlg.isEnded := FALSE;
  				StrAlg.hasError 	:= FALSE;

                                           (*****************       OnReset       *****************)
                                          waitReset(IN:=FALSE);
                                          _resetQuestion1:=FALSE;
                                          _resetQuestion2:=FALSE;
                                          resetPhase(puskOilSystem);
                                          resetPhase(runningEngine);
                                          resetPhase(mvOff);
                                          resetPhase(pnsOn);
                                          resetPhase(wait600);
                                          resetPhase(AutoNUoff);
                                          resetPhase(nu1Off);
                                          resetPhase(nu2Off);
                                          resetPhase(pnsWaitOff);
  	                              resetPhase(autoAvomOff);
                                          resetPhase(Avom1Off);
                                          resetPhase(Avom2Off);
                                          resetPhase(testUnsuccessful);

                                          resetQuestion(questionEngine);
                                          resetQuestion(questionMVoff);

                                          StrAlg.inOpcCommandsDisabled:=FALSE;

  				cmd_for_Status := cmd;
  				source_for_Status := source;
  				command_error_for_Status := 0;
  	END_CASE;
  	resetCmdTimer(IN := false);
  	resetCmdTimerPriznak := TRUE;
  END_IF;
  lastCmd := cmd;

  resetCmdTimer(IN := resetCmdTimerPriznak, PT := T#5S);
  IF resetCmdTimer.Q THEN
  	resetCmdTimerPriznak := FALSE;
  	source_for_Status := 0;
  	cmd_for_Status := 0;
  	command_error_for_Status := 0;
  END_IF;

  StrAlg.Start:= puskOilSystem.startStatus
              OR runningEngine.startStatus
              OR mvOff.startStatus
              OR pnsOn.startStatus
              OR wait600.startStatus
              OR AutoNUoff.startStatus
              OR nu1Off.startStatus
              OR nu2Off.startStatus
              OR pnsWaitOff.startStatus
              OR testUnsuccessful.startStatus;

  StrAlg.Error:=  puskOilSystem.errorStatus
              OR runningEngine.errorStatus
              OR mvOff.errorStatus
              OR pnsOn.errorStatus
              OR wait600.errorStatus
              OR AutoNUoff.errorStatus
              OR nu1Off.errorStatus
              OR nu2Off.errorStatus
              OR pnsWaitOff.errorStatus
              OR testUnsuccessful.errorStatus;

  StrAlg.Top:=   puskOilSystem.topStatus
              OR runningEngine.topStatus
              OR mvOff.topStatus
              OR pnsOn.topStatus
              OR wait600.topStatus
              OR AutoNUoff.topStatus
              OR nu1Off.topStatus
              OR nu2Off.topStatus
              OR pnsWaitOff.topStatus
              OR testUnsuccessful.topStatus;

  (*TODO: TYPE PROGRAM CODE HERE*)
  StrAlg.status :=  SHL(BYTE_TO_DWORD(source_for_Status), 29)
  			OR SHL(BYTE_TO_DWORD(cmd_for_Status), 26)
  			OR SHL(BYTE_TO_DWORD(command_error_for_Status), 23)
  			OR SHL(BOOL_TO_DWORD(StrAlg.OpcCommandsDisabled ), 21)
  			OR SHL(BOOL_TO_DWORD(StrAlg.hasError),4)
  			OR SHL(BOOL_TO_DWORD(StrAlg.CanRun),2)
  			OR SHL(BOOL_TO_DWORD(StrAlg.isEnded),1)
  			OR BOOL_TO_DWORD(StrAlg.isRuning);
END_FUNCTION_BLOCK

FUNCTION_BLOCK testPmsAlg
  VAR_IN_OUT
    StrAlg : struct_Alg;
    algContinue : struct_Question;
  END_VAR
  VAR
    pnsOn : struct_PhaseAlgoritm;
    PmsUp : struct_PhaseAlgoritm;
    runProtecrionAi : struct_PhaseAlgoritm;
    pnsOff : struct_PhaseAlgoritm;
    BreakTest : struct_PhaseAlgoritm;
    LowOilPS : struct_PhaseAlgoritm;
    LowOilAS : struct_PhaseAlgoritm;
    testUnsuccessful : struct_PhaseAlgoritm;
    fb_pnsOn : fb_ph_Switch;
    fb_PmsUp : fb_ph_WaitAnalogValue;
    fb_algContinue : fb_Question;
    fb_runProtecrionAi : fb_ph_AIprotection;
    fb_pnsOff : fb_ph_Switch;
    fb_BreakTest : fb_ph_Timer;
    fb_LowOilPS : fb_ph_CustomPhase;
    fb_LowOilAS : fb_ph_CustomPhase;
    fb_testUnsuccessful : fb_ph_CustomPhase;
    _sunpackerCommand : fb_sunpackerCommand;
    _DualStateImAction : TYPE_DualStateImAction;
    _Answers : TYPE_Answers;
    _statusDualInput : TYPE_statusDualInput;
    _StatusAi : TYPE_StatusAi;
    _PhaseAlgoritmAction : TYPE_PhaseAlgoritmAction;
    source : BYTE;
    cmd : BYTE;
    lastCmd : BYTE;
    source_for_Status : BYTE;
    cmd_for_Status : BYTE;
    command_error_for_Status : BYTE;
    resetCmdTimer : TON;
    resetCmdTimerPriznak : BOOL;
    onInit : BOOL;
    _resetQuestion : BOOL;
    waitReset : TON;
  END_VAR
  VAR_EXTERNAL
    IM : ImConfig;
    algoritms : AlgoritmsConfig;
    ai : AiConfig;
    AlgTimers : struct_AlgTimers;
    ModeGpa : TYPE_ModeGpa;
    algManager : struct_AlgoritmsManager;
    protections : ProtectionsConfig;
  END_VAR

  IF NOT onInit THEN

                     fb_pnsOn(phaseNumber:=0, act:=_on);
          algContinue.AnswerVariants:=_Answers.ANS_YES;
                     fb_PmsUp(phaseNumber:=1);
           fb_runProtecrionAi(phaseNumber:=3, act:=_run);
                    fb_pnsOff(phaseNumber:=4, act:=_off);
                 fb_BreakTest(phaseNumber:=5, delay:=T#120S);
                  fb_LowOilPS(phaseNumber:=6);
                  fb_LowOilAS(phaseNumber:=7);
          fb_testUnsuccessful(phaseNumber:=8);

  onInit:=TRUE;
  END_IF;

              fb_pnsOn(StrPh:=pnsOn, Im:=IM.pns);
        fb_algContinue(StrQ:=algContinue);
              fb_PmsUp(StrPh:=PmsUp, ai:=ai.Pmasla_posle_GNS, more:=ai.Pmasla_posle_GNS.LW);
    fb_runProtecrionAi(StrPh:=runProtecrionAi, StrAiP:=protections.Os_sdvig_nagnetatelja_minus);
             fb_pnsOff(StrPh:=pnsOff, Im:=IM.pns);
          fb_BreakTest(StrPh:=BreakTest, timer:=AlgTimers.testPms_BreakTest);
           fb_LowOilPS(StrPh:=LowOilPS);
           fb_LowOilAS(StrPh:=LowOilAS);
   fb_testUnsuccessful(StrPh:=testUnsuccessful);

  StrAlg.CanRun := StrAlg.inCanRun;
  StrAlg.OpcCommandsDisabled := StrAlg.inOpcCommandsDisabled;

  IF StrAlg.isRuning THEN

      StrAlg.hasError := pnsOn.error OR pnsOff.error OR testUnsuccessful.error;

      IF pnsOn.top THEN
           runPhase(PmsUp);
      END_IF;

      IF PmsUp.top THEN
           runPhase(runProtecrionAi);
      END_IF;

      IF runProtecrionAi.top THEN
           (*IM.SingleSignals.P_oil_low.Disabled_Sig:=FALSE;*)
           ai.Pmasla_posle_GNS.Disabled_LA:=FALSE;
           ai.Pmasla_posle_GNS.Disabled_LW:=FALSE;
           ai.Pmasla_posle_NU.Disabled_LW:=FALSE;
               IF NOT _resetQuestion THEN
                   askQuestion(algContinue);
                   _resetQuestion:=TRUE;
               END_IF;
      END_IF;

      IF algContinue.answer = _Answers.ANS_YES THEN

          runPhase(BreakTest);
          runPhase(pnsOff);
          runPhase(LowOilPS);
          runPhase(LowOilAS);
          resetQuestion(algContinue);

      END_IF;

      IF 	LowOilPS.start AND NOT LowOilPS.top THEN
  	LowOilPS.top:= ai.Pmasla_posle_GNS.interval = _statusAi.LW;
      END_IF;
      IF 	LowOilAS.start AND NOT LowOilAS.top THEN
  	LowOilAS.top:= ai.Pmasla_posle_GNS.interval = _statusAi.LA;
      END_IF;

      IF LowOilPS.top AND LowOilAS.top THEN
            resetPhase(BreakTest);
            waitReset(IN:=TRUE, PT:= T#3S);
      END_IF;

      IF BreakTest.top AND StrAlg.isEnded THEN
  	testUnsuccessful.error:=TRUE;
      END_IF;

      IF waitReset.Q THEN
          algManager.nMode:=ModeGpa.MODE_STOP;
          resetIfRunning(StrAlg);
      END_IF;

      StrAlg.isEnded:= LowOilPS.top AND LowOilAS.top;

  END_IF;

  StrAlg.CanRun := StrAlg.inCanRun;
  StrAlg.OpcCommandsDisabled := StrAlg.inOpcCommandsDisabled;

  (* ---- Если управление с ВУ заблокировано, то  передаем команду из алгоритма ---- *)
  IF StrAlg.inOpcCommandsDisabled THEN
  	StrAlg.inCommand := StrAlg.inCommand_Alg;
  ELSE (* иначе передаем команду с АРМа*)
  	StrAlg.inCommand := StrAlg.inCommand_ARM;
  END_IF;

  _sunpackerCommand(command := StrAlg.inCommand);
  	source := _sunpackerCommand.source;
  	cmd := _sunpackerCommand.cmd;

  IF cmd <> 0 AND lastCmd <> cmd AND (((NOT StrAlg.opcCommandsDisabled) AND source > 0) OR source = 0) then
  	CASE BYTE_TO_INT(cmd) OF
  		(*cmdRun*) 1: 	IF (StrAlg.CanRun) THEN
  					StrAlg.isRuning := TRUE;
  					StrAlg.isEnded := FALSE;
  					StrAlg.hasError := FALSE;
  					(*****************       OnRun       *****************)

                                                    algManager.nMode:=ModeGpa.MODE_TESTPMS;
                                                    resetAndDisable(alg:=algoritms.ppu);
                                                    runPhase(pnsOn);

  					cmd_for_Status := cmd;
  					source_for_Status := source;
  					command_error_for_Status := 0;
  				ELSE
  					StrAlg.isRuning := FALSE;
  					StrAlg.isEnded := FALSE;
  					StrAlg.hasError 	:= FALSE;

  					cmd_for_Status := 0;
  					source_for_Status := source;
  					command_error_for_Status := cmd;
  				END_IF;
  		(*cmdReset*) 2: 	StrAlg.isRuning := FALSE;
  				StrAlg.isEnded := FALSE;
  				StrAlg.hasError 	:= FALSE;

                                           (*****************       OnReset       *****************)
                                          waitReset(IN:=FALSE);
                                          _resetQuestion:=FALSE;
                                          ai.Pmasla_posle_GNS.Disabled_LA:=TRUE;
                                          ai.Pmasla_posle_GNS.Disabled_LW:=TRUE;
                                          ai.Pmasla_posle_NU.Disabled_LW:=TRUE;
                                         (* IM.SingleSignals.P_oil_low.Disabled_Sig:=TRUE;*)
                                          resetAiProtection(protections.Os_sdvig_nagnetatelja_minus);

                                          resetPhase(pnsOn);
                                          resetPhase(PmsUp);
                                          resetPhase(runProtecrionAi);
                                          resetPhase(pnsOff);
                                          resetPhase(BreakTest);
                                          resetPhase(LowOilPS);
                                          resetPhase(LowOilAS);
                                          resetPhase(testUnsuccessful);

                                          resetQuestion(algContinue);

                                          StrAlg.inOpcCommandsDisabled:=FALSE;

  				cmd_for_Status := cmd;
  				source_for_Status := source;
  				command_error_for_Status := 0;
  	END_CASE;
  	resetCmdTimer(IN := false);
  	resetCmdTimerPriznak := TRUE;
  END_IF;
  lastCmd := cmd;

  resetCmdTimer(IN := resetCmdTimerPriznak, PT := T#5S);
  IF resetCmdTimer.Q THEN
  	resetCmdTimerPriznak := FALSE;
  	source_for_Status := 0;
  	cmd_for_Status := 0;
  	command_error_for_Status := 0;
  END_IF;

  StrAlg.Start:= pnsOn.startStatus
              OR PmsUp.startStatus
              OR runProtecrionAi.startStatus
              OR pnsOff.startStatus
              OR BreakTest.startStatus
              OR LowOilPS.startStatus
              OR LowOilAS.startStatus
              OR testUnsuccessful.startStatus;

  StrAlg.Error:= pnsOn.errorStatus
              OR PmsUp.errorStatus
              OR runProtecrionAi.errorStatus
              OR pnsOff.errorStatus
              OR BreakTest.errorStatus
              OR LowOilPS.errorStatus
              OR LowOilAS.errorStatus
              OR testUnsuccessful.errorStatus;

  StrAlg.Top:=   pnsOn.topStatus
              OR PmsUp.topStatus
              OR runProtecrionAi.topStatus
              OR pnsOff.topStatus
              OR BreakTest.topStatus
              OR LowOilPS.topStatus
              OR LowOilAS.topStatus
              OR testUnsuccessful.topStatus;

  (*TODO: TYPE PROGRAM CODE HERE*)
  StrAlg.status :=  SHL(BYTE_TO_DWORD(source_for_Status), 29)
  			OR SHL(BYTE_TO_DWORD(cmd_for_Status), 26)
  			OR SHL(BYTE_TO_DWORD(command_error_for_Status), 23)
  			OR SHL(BOOL_TO_DWORD(StrAlg.OpcCommandsDisabled ), 21)
  			OR SHL(BOOL_TO_DWORD(StrAlg.hasError),4)
  			OR SHL(BOOL_TO_DWORD(StrAlg.CanRun),2)
  			OR SHL(BOOL_TO_DWORD(StrAlg.isEnded),1)
  			OR BOOL_TO_DWORD(StrAlg.isRuning);
END_FUNCTION_BLOCK

FUNCTION_BLOCK ApuskAlg
  VAR_IN_OUT
    StrAlg : struct_Alg;
  END_VAR
  VAR
    runOilsystem : struct_PhaseAlgoritm;
    runEngine : struct_PhaseAlgoritm;
    filling : struct_PhaseAlgoritm;
    fb_runOilsystem : fb_ph_algoritm;
    fb_runEngine : fb_ph_algoritm;
    fb_filling : fb_ph_algoritm;
    _sunpackerCommand : fb_sunpackerCommand;
    _PhaseAlgoritmAction : TYPE_PhaseAlgoritmAction;
    _statusDualInput : TYPE_statusDualInput;
    source : BYTE;
    cmd : BYTE;
    lastCmd : BYTE;
    source_for_Status : BYTE;
    cmd_for_Status : BYTE;
    command_error_for_Status : BYTE;
    resetCmdTimer : TON;
    resetCmdTimerPriznak : BOOL;
    onInit : BOOL;
    waitReset : TON;
  END_VAR
  VAR_EXTERNAL
    algoritms : AlgoritmsConfig;
    ModeGpa : TYPE_ModeGpa;
    algManager : struct_AlgoritmsManager;
    IM : ImConfig;
  END_VAR

  IF NOT onInit THEN

           fb_runOilsystem(phaseNumber:=0, act:=_run, waitCompletion:=TRUE);
              fb_runEngine(phaseNumber:=1, act:=_run, waitCompletion:=TRUE);
                fb_filling(phaseNumber:=2, act:=_run, waitCompletion:=TRUE);

  onInit:=TRUE;
  END_IF;

           fb_runOilsystem(StrPh:=runOilsystem, alg:=algoritms.puskOilSystem);
              fb_runEngine(StrPh:=runEngine, alg:=algoritms.engineRun);
                fb_filling(StrPh:=filling, alg:=algoritms.filling);

  StrAlg.CanRun := StrAlg.inCanRun;
  StrAlg.OpcCommandsDisabled := StrAlg.inOpcCommandsDisabled;

  IF StrAlg.isRuning THEN

      StrAlg.hasError := runOilsystem.error OR runEngine.error OR filling.error;

      IF runOilsystem.top THEN
           runPhase(runEngine);
      END_IF;

      IF runEngine.top THEN
           runPhase(filling);
      END_IF;

      IF filling.top THEN
            waitReset(IN:=TRUE, PT:= T#2S);
      END_IF;

      IF waitReset.Q THEN

          IF Im.kran6.onStatus = _statusDualInput.STATUS_On THEN
  	algManager.nMode:= ModeGpa.MODE_WORK_Ring;
          END_IF;
          IF Im.kran6.onStatus = _statusDualInput.STATUS_Off THEN
  	algManager.nMode:= ModeGpa.MODE_WORK_Line;
          END_IF;

          resetIfRunning(StrAlg);
      END_IF;

      StrAlg.isEnded:= filling.top;

  END_IF;

  StrAlg.CanRun := StrAlg.inCanRun;
  StrAlg.OpcCommandsDisabled := StrAlg.inOpcCommandsDisabled;

  (* ---- Если управление с ВУ заблокировано, то  передаем команду из алгоритма ---- *)
  IF StrAlg.inOpcCommandsDisabled THEN
  	StrAlg.inCommand := StrAlg.inCommand_Alg;
  ELSE (* иначе передаем команду с АРМа*)
  	StrAlg.inCommand := StrAlg.inCommand_ARM;
  END_IF;

  _sunpackerCommand(command := StrAlg.inCommand);
  	source := _sunpackerCommand.source;
  	cmd := _sunpackerCommand.cmd;

  IF cmd <> 0 AND lastCmd <> cmd AND (((NOT StrAlg.opcCommandsDisabled) AND source > 0) OR source = 0) then
  	CASE BYTE_TO_INT(cmd) OF
  		(*cmdRun*) 1: 	IF (StrAlg.CanRun) THEN
  					StrAlg.isRuning := TRUE;
  					StrAlg.isEnded := FALSE;
  					StrAlg.hasError := FALSE;
  					(*****************       OnRun       *****************)

                                                    algoritms.puskOilSystem.inCanRun:= TRUE	;
                                                    algoritms.filling.inCanRun:= TRUE	;
                                                    algoritms.engineRun.inCanRun:= TRUE	;

                                                    algManager.nMode:=ModeGpa.MODE_APUSK;
                                                    (*impulseSO(Im.SingleOutputs.VzvodBREO);*)
                                                    runPhase(runOilsystem);

  					cmd_for_Status := cmd;
  					source_for_Status := source;
  					command_error_for_Status := 0;
  				ELSE
  					StrAlg.isRuning := FALSE;
  					StrAlg.isEnded := FALSE;
  					StrAlg.hasError 	:= FALSE;

  					cmd_for_Status := 0;
  					source_for_Status := source;
  					command_error_for_Status := cmd;
  				END_IF;
  		(*cmdReset*) 2: 	StrAlg.isRuning := FALSE;
  				StrAlg.isEnded := FALSE;
  				StrAlg.hasError 	:= FALSE;

                                           (*****************       OnReset       *****************)
                                          waitReset(IN:=FALSE);
                                          StrAlg.inCanRun:=FALSE;

                                          resetPhase(runOilsystem);
                                          resetPhase(runEngine);
                                          resetPhase(filling);

                                          StrAlg.inOpcCommandsDisabled:=FALSE;

  				cmd_for_Status := cmd;
  				source_for_Status := source;
  				command_error_for_Status := 0;
  	END_CASE;
  	resetCmdTimer(IN := false);
  	resetCmdTimerPriznak := TRUE;
  END_IF;
  lastCmd := cmd;

  resetCmdTimer(IN := resetCmdTimerPriznak, PT := T#5S);
  IF resetCmdTimer.Q THEN
  	resetCmdTimerPriznak := FALSE;
  	source_for_Status := 0;
  	cmd_for_Status := 0;
  	command_error_for_Status := 0;
  END_IF;

  StrAlg.Start:= runOilsystem.startStatus
              OR runEngine.startStatus
              OR filling.startStatus;

  StrAlg.Error:= runOilsystem.errorStatus
              OR runEngine.errorStatus
              OR filling.errorStatus;

  StrAlg.Top:=   runOilsystem.topStatus
              OR runEngine.topStatus
              OR filling.topStatus;

  (*TODO: TYPE PROGRAM CODE HERE*)
  StrAlg.status :=  SHL(BYTE_TO_DWORD(source_for_Status), 29)
  			OR SHL(BYTE_TO_DWORD(cmd_for_Status), 26)
  			OR SHL(BYTE_TO_DWORD(command_error_for_Status), 23)
  			OR SHL(BOOL_TO_DWORD(StrAlg.OpcCommandsDisabled ), 21)
  			OR SHL(BOOL_TO_DWORD(StrAlg.hasError),4)
  			OR SHL(BOOL_TO_DWORD(StrAlg.CanRun),2)
  			OR SHL(BOOL_TO_DWORD(StrAlg.isEnded),1)
  			OR BOOL_TO_DWORD(StrAlg.isRuning);
END_FUNCTION_BLOCK

FUNCTION_BLOCK Pusk_first_faza1
  VAR_IN_OUT
    StrAlg : struct_Alg;
  END_VAR
  VAR
    timer240 : struct_PhaseAlgoritm;
    pmsMore50 : struct_PhaseAlgoritm;
    pnsOn : struct_PhaseAlgoritm;
    pmsMore300 : struct_PhaseAlgoritm;
    Protection_Pms : struct_PhaseAlgoritm;
    Error_Alg : struct_PhaseAlgoritm;
    fb_timer240 : fb_ph_Timer;
    fb_PnmMore50 : fb_ph_algoritm;
    fb_PnsOn : fb_ph_Switch;
    fb_PmsMore300 : fb_ph_algoritm;
    fb_Protection_Pms : fb_ph_algoritm;
    fb_Error_Alg : fb_ph_algoritm;
    _sunpackerCommand : fb_sunpackerCommand;
    _PhaseAlgoritmAction : TYPE_PhaseAlgoritmAction;
    _statusDualInput : TYPE_statusDualInput;
    _Answers : TYPE_Answers;
    source : BYTE;
    cmd : BYTE;
    lastCmd : BYTE;
    source_for_Status : BYTE;
    cmd_for_Status : BYTE;
    command_error_for_Status : BYTE;
    resetCmdTimer : TON;
    resetCmdTimerPriznak : BOOL;
    onInit : BOOL;
    waitReset : TON;
  END_VAR
  VAR_EXTERNAL
    ModeGpa : TYPE_ModeGpa;
    algManager : struct_AlgoritmsManager;
    IM : ImConfig;
    protections : ProtectionsConfig;
  END_VAR
  VAR
    _statusAi : TYPE_StatusAi;
  END_VAR
  VAR_EXTERNAL
    ai : AiConfig;
  END_VAR

  IF NOT onInit THEN

           fb_timer240(phaseNumber:=0, delay:=T#240S);
           fb_PnmMore50(phaseNumber:=1);
           fb_PnsOn(phaseNumber:=2, act:=_on);
           fb_PmsMore300(phaseNumber:=3);
           fb_Protection_Pms(phaseNumber:=4);
           fb_Error_Alg(phaseNumber:=5);

  onInit:=TRUE;
  END_IF;
